REGION Network 62: Falownik P4
   // Sterowaniem pracy z falownika. Sterowanie napędem na pozycji MC
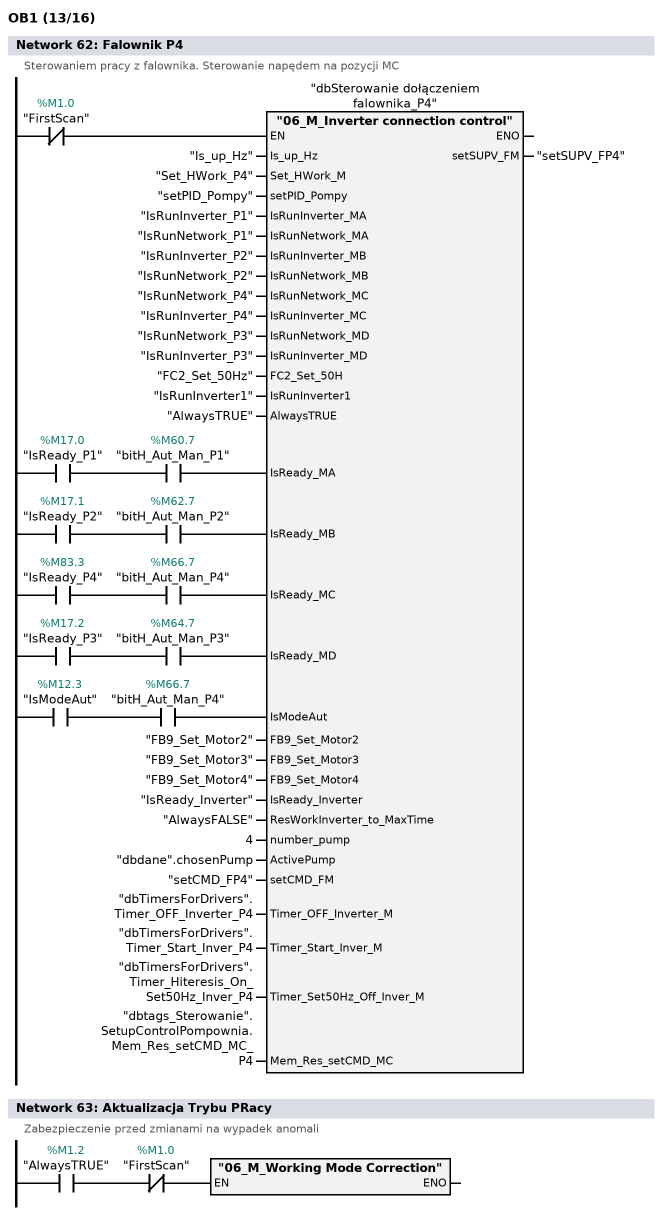
   RUNG wire#powerrail
      I_Contact( "FirstScan" )
      "dbSterowanie dołączeniem falownika_P4"(IsReady_MA := wire#w1, IsReady_MB := wire#w2, IsReady_MC := wire#w3, IsReady_MD := wire#w4, IsModeAut := wire#w5, Is_up_Hz := "Is_up_Hz", Set_HWork_M := "Set_HWork_P4", setPID_Pompy := "setPID_Pompy", IsRunInverter_MA := "IsRunInverter_P1", IsRunNetwork_MA := "IsRunNetwork_P1", IsRunInverter_MB := "IsRunInverter_P2", IsRunNetwork_MB := "IsRunNetwork_P2", IsRunNetwork_MC := "IsRunNetwork_P4", IsRunInverter_MC := "IsRunInverter_P4", IsRunNetwork_MD := "IsRunNetwork_P3", IsRunInverter_MD := "IsRunInverter_P3", FC2_Set_50H := "FC2_Set_50Hz", IsRunInverter1 := "IsRunInverter1", AlwaysTRUE := "AlwaysTRUE", FB9_Set_Motor2 := "FB9_Set_Motor2", FB9_Set_Motor3 := "FB9_Set_Motor3", FB9_Set_Motor4 := "FB9_Set_Motor4", IsReady_Inverter := "IsReady_Inverter", ResWorkInverter_to_MaxTime := "AlwaysFALSE", number_pump := 4, ActivePump := "dbdane".chosenPump, setCMD_FM := "setCMD_FP4", Timer_OFF_Inverter_M := "dbTimersForDrivers".Timer_OFF_Inverter_P4, Timer_Start_Inver_M := "dbTimersForDrivers".Timer_Start_Inver_P4, Timer_Set50Hz_Off_Inver_M := "dbTimersForDrivers".Timer_Hiteresis_On_Set50Hz_Inver_P4, Mem_Res_setCMD_MC := "dbtags_Sterowanie".SetupControlPompownia.Mem_Res_setCMD_MC_P4, setSUPV_FM => "setSUPV_FP4")
   END_RUNG
   RUNG wire#powerrail
      Contact( "IsReady_P1" )
      Contact( "bitH_Aut_Man_P1" )
   END_RUNG wire#w1
   RUNG wire#powerrail
      Contact( "IsReady_P2" )
      Contact( "bitH_Aut_Man_P2" )
   END_RUNG wire#w2
   RUNG wire#powerrail
      Contact( "IsReady_P4" )
      Contact( "bitH_Aut_Man_P4" )
   END_RUNG wire#w3
   RUNG wire#powerrail
      Contact( "IsReady_P3" )
      Contact( "bitH_Aut_Man_P3" )
   END_RUNG wire#w4
   RUNG wire#powerrail
      Contact( "IsModeAut" )
      Contact( "bitH_Aut_Man_P4" )
   END_RUNG wire#w5
   // the same network as SCL:
   IF NOT "FirstScan" THEN
       "dbSterowanie dołączeniem falownika_P4"(Is_up_Hz := "Is_up_Hz",   // "06_M_Inverter connection control"
                               Set_HWork_M := "Set_HWork_P4",
                               setPID_Pompy := "setPID_Pompy",
                               IsRunInverter_MA := "IsRunInverter_P1",
                               IsRunNetwork_MA := "IsRunNetwork_P1",
                               IsRunInverter_MB := "IsRunInverter_P2",
                               IsRunNetwork_MB := "IsRunNetwork_P2",
                               IsRunNetwork_MC := "IsRunNetwork_P4",
                               IsRunInverter_MC := "IsRunInverter_P4",
                               IsRunNetwork_MD := "IsRunNetwork_P3",
                               IsRunInverter_MD := "IsRunInverter_P3",
                               FC2_Set_50H := "FC2_Set_50Hz",
                               IsRunInverter1 := "IsRunInverter1",
                               AlwaysTRUE := "AlwaysTRUE",
                               IsReady_MA := "IsReady_P1" AND "bitH_Aut_Man_P1",
                               IsReady_MB := "IsReady_P2" AND "bitH_Aut_Man_P2",
                               IsReady_MC := "IsReady_P4" AND "bitH_Aut_Man_P4",
                               IsReady_MD := "IsReady_P3" AND "bitH_Aut_Man_P3",
                               IsModeAut := "IsModeAut" AND "bitH_Aut_Man_P4",
                               FB9_Set_Motor2 := "FB9_Set_Motor2",
                               FB9_Set_Motor3 := "FB9_Set_Motor3",
                               FB9_Set_Motor4 := "FB9_Set_Motor4",
                               IsReady_Inverter := "IsReady_Inverter",
                               ResWorkInverter_to_MaxTime := "AlwaysFALSE",
                               number_pump := 4,
                               ActivePump := "dbdane".chosenPump,
                               setCMD_FM := "setCMD_FP4",
                               Timer_OFF_Inverter_M := "dbTimersForDrivers".Timer_OFF_Inverter_P4,
                               Timer_Start_Inver_M := "dbTimersForDrivers".Timer_Start_Inver_P4,
                               Timer_Set50Hz_Off_Inver_M := "dbTimersForDrivers".Timer_Hiteresis_On_Set50Hz_Inver_P4,
                               Mem_Res_setCMD_MC := "dbtags_Sterowanie".SetupControlPompownia.Mem_Res_setCMD_MC_P4,
                               setSUPV_FM => "setSUPV_FP4");
   END_IF;
END_REGION

REGION Network 63: Aktualizacja Trybu PRacy
   // Zabezpieczenie przed zmianami na wypadek anomali
   RUNG wire#powerrail
      Contact( "AlwaysTRUE" )
      I_Contact( "FirstScan" )
      "06_M_Working Mode Correction"()
   END_RUNG
   // the same network as SCL:
   IF "AlwaysTRUE" AND NOT "FirstScan" THEN "06_M_Working Mode Correction"(); END_IF;
END_REGION

REGION Network 64: Sterowanie falownikiem
   // Sterowanie załaczaniem falownika
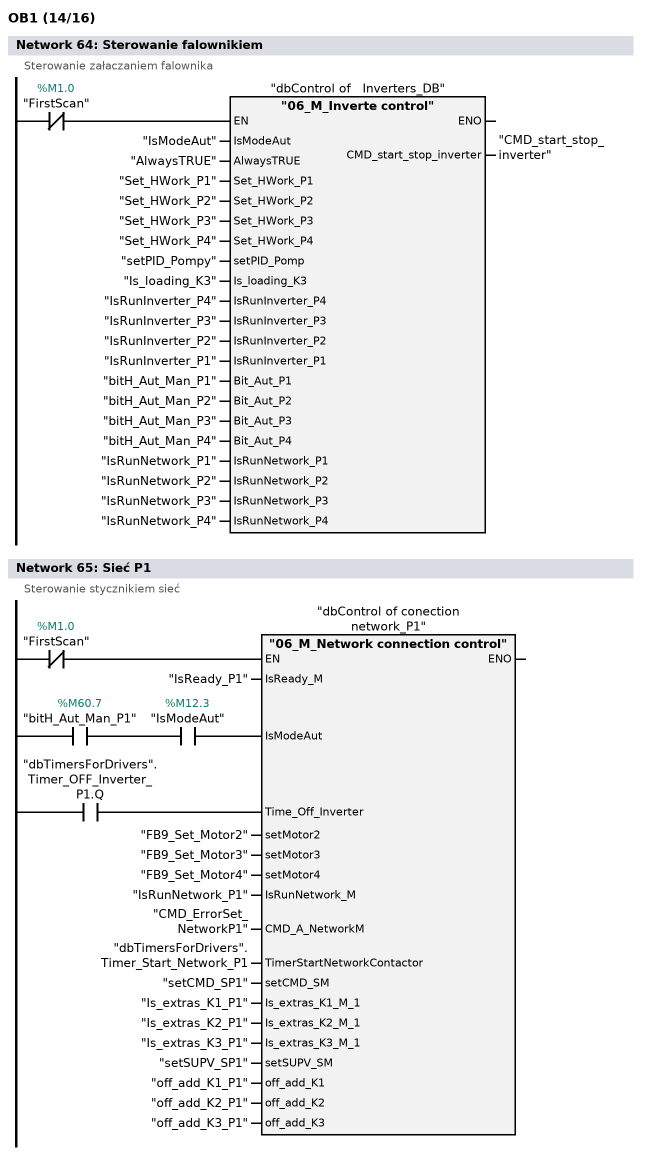
   RUNG wire#powerrail
      I_Contact( "FirstScan" )
      "dbControl of   Inverters_DB"(IsModeAut := "IsModeAut", AlwaysTRUE := "AlwaysTRUE", Set_HWork_P1 := "Set_HWork_P1", Set_HWork_P2 := "Set_HWork_P2", Set_HWork_P3 := "Set_HWork_P3", Set_HWork_P4 := "Set_HWork_P4", setPID_Pomp := "setPID_Pompy", Is_loading_K3 := "Is_loading_K3", IsRunInverter_P4 := "IsRunInverter_P4", IsRunInverter_P3 := "IsRunInverter_P3", IsRunInverter_P2 := "IsRunInverter_P2", IsRunInverter_P1 := "IsRunInverter_P1", Bit_Aut_P1 := "bitH_Aut_Man_P1", Bit_Aut_P2 := "bitH_Aut_Man_P2", Bit_Aut_P3 := "bitH_Aut_Man_P3", Bit_Aut_P4 := "bitH_Aut_Man_P4", IsRunNetwork_P1 := "IsRunNetwork_P1", IsRunNetwork_P2 := "IsRunNetwork_P2", IsRunNetwork_P3 := "IsRunNetwork_P3", IsRunNetwork_P4 := "IsRunNetwork_P4", CMD_start_stop_inverter => "CMD_start_stop_inverter")
   END_RUNG
   // the same network as SCL:
   IF NOT "FirstScan" THEN
       "dbControl of   Inverters_DB"(IsModeAut := "IsModeAut",   // "06_M_Inverte control"
                               AlwaysTRUE := "AlwaysTRUE",
                               Set_HWork_P1 := "Set_HWork_P1",
                               Set_HWork_P2 := "Set_HWork_P2",
                               Set_HWork_P3 := "Set_HWork_P3",
                               Set_HWork_P4 := "Set_HWork_P4",
                               setPID_Pomp := "setPID_Pompy",
                               Is_loading_K3 := "Is_loading_K3",
                               IsRunInverter_P4 := "IsRunInverter_P4",
                               IsRunInverter_P3 := "IsRunInverter_P3",
                               IsRunInverter_P2 := "IsRunInverter_P2",
                               IsRunInverter_P1 := "IsRunInverter_P1",
                               Bit_Aut_P1 := "bitH_Aut_Man_P1",
                               Bit_Aut_P2 := "bitH_Aut_Man_P2",
                               Bit_Aut_P3 := "bitH_Aut_Man_P3",
                               Bit_Aut_P4 := "bitH_Aut_Man_P4",
                               IsRunNetwork_P1 := "IsRunNetwork_P1",
                               IsRunNetwork_P2 := "IsRunNetwork_P2",
                               IsRunNetwork_P3 := "IsRunNetwork_P3",
                               IsRunNetwork_P4 := "IsRunNetwork_P4",
                               CMD_start_stop_inverter => "CMD_start_stop_inverter");
   END_IF;
END_REGION

REGION Network 65: Sieć P1
   // Sterowanie stycznikiem sieć
   RUNG wire#powerrail
      I_Contact( "FirstScan" )
      "dbControl of conection network_P1"(IsModeAut := wire#w1, Time_Off_Inverter := wire#w2, IsReady_M := "IsReady_P1", setMotor2 := "FB9_Set_Motor2", setMotor3 := "FB9_Set_Motor3", setMotor4 := "FB9_Set_Motor4", IsRunNetwork_M := "IsRunNetwork_P1", CMD_A_NetworkM := "CMD_ErrorSet_NetworkP1", TimerStartNetworkContactor := "dbTimersForDrivers".Timer_Start_Network_P1, setCMD_SM := "setCMD_SP1", Is_extras_K1_M_1 := "Is_extras_K1_P1", Is_extras_K2_M_1 := "Is_extras_K2_P1", Is_extras_K3_M_1 := "Is_extras_K3_P1", setSUPV_SM := "setSUPV_SP1", off_add_K1 := "off_add_K1_P1", off_add_K2 := "off_add_K2_P1", off_add_K3 := "off_add_K3_P1")
   END_RUNG
   RUNG wire#powerrail
      Contact( "bitH_Aut_Man_P1" )
      Contact( "IsModeAut" )
   END_RUNG wire#w1
   RUNG wire#powerrail
      Contact( "dbTimersForDrivers".Timer_OFF_Inverter_P1.Q )
   END_RUNG wire#w2
   // the same network as SCL:
   IF NOT "FirstScan" THEN
       "dbControl of conection network_P1"(IsReady_M := "IsReady_P1",   // "06_M_Network connection control"
                               IsModeAut := "bitH_Aut_Man_P1" AND "IsModeAut",
                               Time_Off_Inverter := "dbTimersForDrivers".Timer_OFF_Inverter_P1.Q,
                               setMotor2 := "FB9_Set_Motor2",
                               setMotor3 := "FB9_Set_Motor3",
                               setMotor4 := "FB9_Set_Motor4",
                               IsRunNetwork_M := "IsRunNetwork_P1",
                               CMD_A_NetworkM := "CMD_ErrorSet_NetworkP1",
                               TimerStartNetworkContactor := "dbTimersForDrivers".Timer_Start_Network_P1,
                               setCMD_SM := "setCMD_SP1",
                               Is_extras_K1_M_1 := "Is_extras_K1_P1",
                               Is_extras_K2_M_1 := "Is_extras_K2_P1",
                               Is_extras_K3_M_1 := "Is_extras_K3_P1",
                               setSUPV_SM := "setSUPV_SP1",
                               off_add_K1 := "off_add_K1_P1",
                               off_add_K2 := "off_add_K2_P1",
                               off_add_K3 := "off_add_K3_P1");
   END_IF;
END_REGION

REGION Network 66: Sieć P2
   // Sterowanie stycznikiem sieć
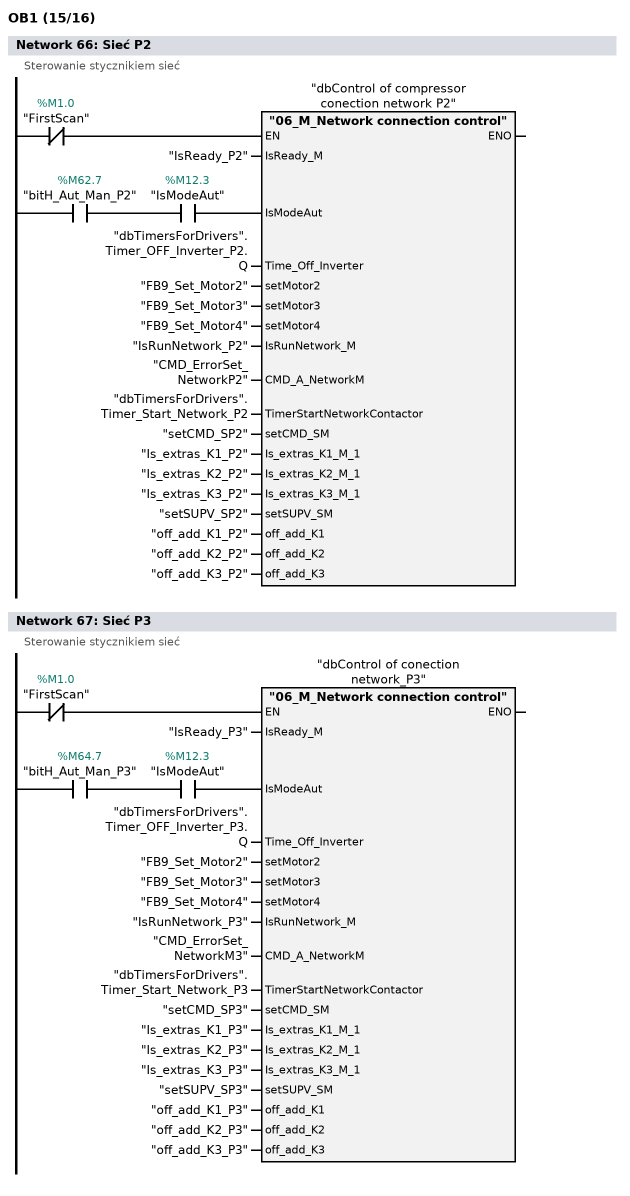
   RUNG wire#powerrail
      I_Contact( "FirstScan" )
      "dbControl of compressor conection network P2"(IsModeAut := wire#w1, IsReady_M := "IsReady_P2", Time_Off_Inverter := "dbTimersForDrivers".Timer_OFF_Inverter_P2.Q, setMotor2 := "FB9_Set_Motor2", setMotor3 := "FB9_Set_Motor3", setMotor4 := "FB9_Set_Motor4", IsRunNetwork_M := "IsRunNetwork_P2", CMD_A_NetworkM := "CMD_ErrorSet_NetworkP2", TimerStartNetworkContactor := "dbTimersForDrivers".Timer_Start_Network_P2, setCMD_SM := "setCMD_SP2", Is_extras_K1_M_1 := "Is_extras_K1_P2", Is_extras_K2_M_1 := "Is_extras_K2_P2", Is_extras_K3_M_1 := "Is_extras_K3_P2", setSUPV_SM := "setSUPV_SP2", off_add_K1 := "off_add_K1_P2", off_add_K2 := "off_add_K2_P2", off_add_K3 := "off_add_K3_P2")
   END_RUNG
   RUNG wire#powerrail
      Contact( "bitH_Aut_Man_P2" )
      Contact( "IsModeAut" )
   END_RUNG wire#w1
   // the same network as SCL:
   IF NOT "FirstScan" THEN
       "dbControl of compressor conection network P2"(IsReady_M := "IsReady_P2",   // "06_M_Network connection control"
                               IsModeAut := "bitH_Aut_Man_P2" AND "IsModeAut",
                               Time_Off_Inverter := "dbTimersForDrivers".Timer_OFF_Inverter_P2.Q,
                               setMotor2 := "FB9_Set_Motor2",
                               setMotor3 := "FB9_Set_Motor3",
                               setMotor4 := "FB9_Set_Motor4",
                               IsRunNetwork_M := "IsRunNetwork_P2",
                               CMD_A_NetworkM := "CMD_ErrorSet_NetworkP2",
                               TimerStartNetworkContactor := "dbTimersForDrivers".Timer_Start_Network_P2,
                               setCMD_SM := "setCMD_SP2",
                               Is_extras_K1_M_1 := "Is_extras_K1_P2",
                               Is_extras_K2_M_1 := "Is_extras_K2_P2",
                               Is_extras_K3_M_1 := "Is_extras_K3_P2",
                               setSUPV_SM := "setSUPV_SP2",
                               off_add_K1 := "off_add_K1_P2",
                               off_add_K2 := "off_add_K2_P2",
                               off_add_K3 := "off_add_K3_P2");
   END_IF;
END_REGION

REGION Network 67: Sieć P3
   // Sterowanie stycznikiem sieć
   RUNG wire#powerrail
      I_Contact( "FirstScan" )
      "dbControl of conection network_P3"(IsModeAut := wire#w1, IsReady_M := "IsReady_P3", Time_Off_Inverter := "dbTimersForDrivers".Timer_OFF_Inverter_P3.Q, setMotor2 := "FB9_Set_Motor2", setMotor3 := "FB9_Set_Motor3", setMotor4 := "FB9_Set_Motor4", IsRunNetwork_M := "IsRunNetwork_P3", CMD_A_NetworkM := "CMD_ErrorSet_NetworkM3", TimerStartNetworkContactor := "dbTimersForDrivers".Timer_Start_Network_P3, setCMD_SM := "setCMD_SP3", Is_extras_K1_M_1 := "Is_extras_K1_P3", Is_extras_K2_M_1 := "Is_extras_K2_P3", Is_extras_K3_M_1 := "Is_extras_K3_P3", setSUPV_SM := "setSUPV_SP3", off_add_K1 := "off_add_K1_P3", off_add_K2 := "off_add_K2_P3", off_add_K3 := "off_add_K3_P3")
   END_RUNG
   RUNG wire#powerrail
      Contact( "bitH_Aut_Man_P3" )
      Contact( "IsModeAut" )
   END_RUNG wire#w1
   // the same network as SCL:
   IF NOT "FirstScan" THEN
       "dbControl of conection network_P3"(IsReady_M := "IsReady_P3",   // "06_M_Network connection control"
                               IsModeAut := "bitH_Aut_Man_P3" AND "IsModeAut",
                               Time_Off_Inverter := "dbTimersForDrivers".Timer_OFF_Inverter_P3.Q,
                               setMotor2 := "FB9_Set_Motor2",
                               setMotor3 := "FB9_Set_Motor3",
                               setMotor4 := "FB9_Set_Motor4",
                               IsRunNetwork_M := "IsRunNetwork_P3",
                               CMD_A_NetworkM := "CMD_ErrorSet_NetworkM3",
                               TimerStartNetworkContactor := "dbTimersForDrivers".Timer_Start_Network_P3,
                               setCMD_SM := "setCMD_SP3",
                               Is_extras_K1_M_1 := "Is_extras_K1_P3",
                               Is_extras_K2_M_1 := "Is_extras_K2_P3",
                               Is_extras_K3_M_1 := "Is_extras_K3_P3",
                               setSUPV_SM := "setSUPV_SP3",
                               off_add_K1 := "off_add_K1_P3",
                               off_add_K2 := "off_add_K2_P3",
                               off_add_K3 := "off_add_K3_P3");
   END_IF;
END_REGION

REGION Network 68: Sieć P4
   // !!!!!!!!!!!!!!!!!!!!! ------------------ Brak pompy --------------------------!!!!!!!!!!!!!!!!!!!!!!!!!!!!!!!
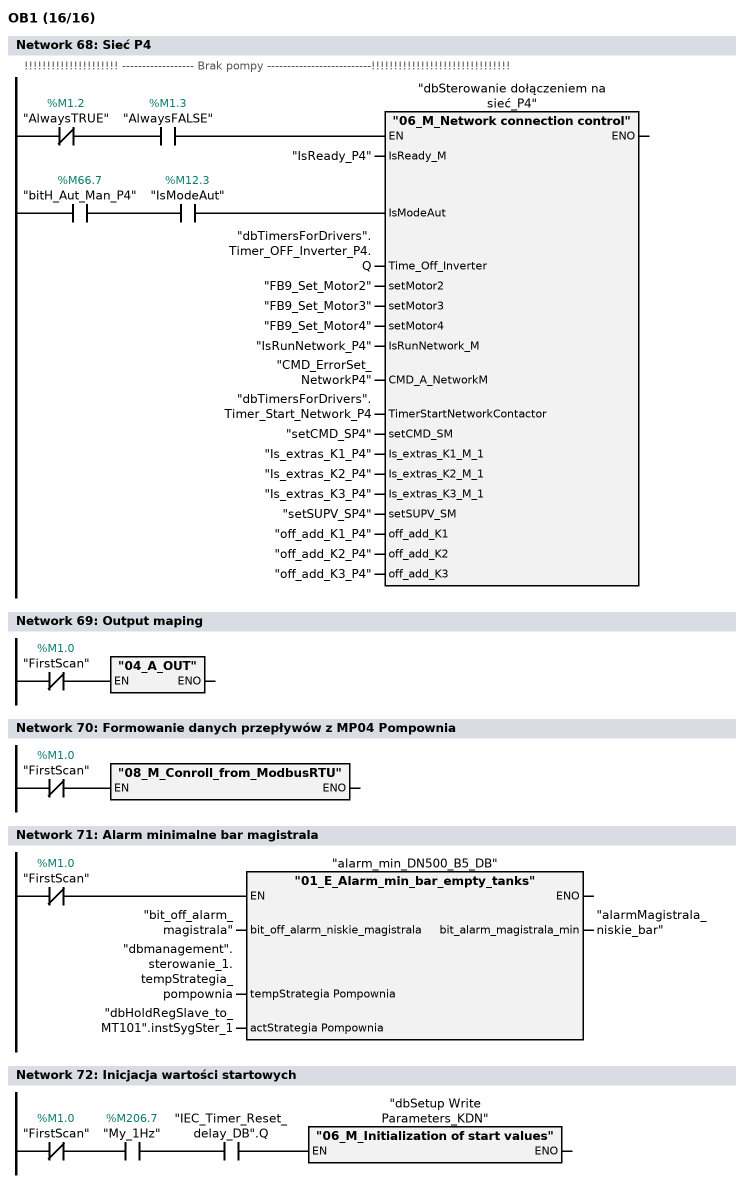
   RUNG wire#powerrail
      I_Contact( "AlwaysTRUE" )
      Contact( "AlwaysFALSE" )
      "dbSterowanie dołączeniem na sieć_P4"(IsModeAut := wire#w1, IsReady_M := "IsReady_P4", Time_Off_Inverter := "dbTimersForDrivers".Timer_OFF_Inverter_P4.Q, setMotor2 := "FB9_Set_Motor2", setMotor3 := "FB9_Set_Motor3", setMotor4 := "FB9_Set_Motor4", IsRunNetwork_M := "IsRunNetwork_P4", CMD_A_NetworkM := "CMD_ErrorSet_NetworkP4", TimerStartNetworkContactor := "dbTimersForDrivers".Timer_Start_Network_P4, setCMD_SM := "setCMD_SP4", Is_extras_K1_M_1 := "Is_extras_K1_P4", Is_extras_K2_M_1 := "Is_extras_K2_P4", Is_extras_K3_M_1 := "Is_extras_K3_P4", setSUPV_SM := "setSUPV_SP4", off_add_K1 := "off_add_K1_P4", off_add_K2 := "off_add_K2_P4", off_add_K3 := "off_add_K3_P4")
   END_RUNG
   RUNG wire#powerrail
      Contact( "bitH_Aut_Man_P4" )
      Contact( "IsModeAut" )
   END_RUNG wire#w1
   // the same network as SCL:
   IF NOT "AlwaysTRUE" AND "AlwaysFALSE" THEN
       "dbSterowanie dołączeniem na sieć_P4"(IsReady_M := "IsReady_P4",   // "06_M_Network connection control"
                               IsModeAut := "bitH_Aut_Man_P4" AND "IsModeAut",
                               Time_Off_Inverter := "dbTimersForDrivers".Timer_OFF_Inverter_P4.Q,
                               setMotor2 := "FB9_Set_Motor2",
                               setMotor3 := "FB9_Set_Motor3",
                               setMotor4 := "FB9_Set_Motor4",
                               IsRunNetwork_M := "IsRunNetwork_P4",
                               CMD_A_NetworkM := "CMD_ErrorSet_NetworkP4",
                               TimerStartNetworkContactor := "dbTimersForDrivers".Timer_Start_Network_P4,
                               setCMD_SM := "setCMD_SP4",
                               Is_extras_K1_M_1 := "Is_extras_K1_P4",
                               Is_extras_K2_M_1 := "Is_extras_K2_P4",
                               Is_extras_K3_M_1 := "Is_extras_K3_P4",
                               setSUPV_SM := "setSUPV_SP4",
                               off_add_K1 := "off_add_K1_P4",
                               off_add_K2 := "off_add_K2_P4",
                               off_add_K3 := "off_add_K3_P4");
   END_IF;
END_REGION

REGION Network 69: Output maping
   RUNG wire#powerrail
      I_Contact( "FirstScan" )
      "04_A_OUT"()
   END_RUNG
   // the same network as SCL:
   IF NOT "FirstScan" THEN "04_A_OUT"(); END_IF;
END_REGION

REGION Network 70: Formowanie danych przepływów z MP04 Pompownia
   RUNG wire#powerrail
      I_Contact( "FirstScan" )
      "08_M_Conroll_from_ModbusRTU"()
   END_RUNG
   // the same network as SCL:
   IF NOT "FirstScan" THEN "08_M_Conroll_from_ModbusRTU"(); END_IF;
END_REGION

REGION Network 71: Alarm minimalne bar magistrala
   RUNG wire#powerrail
      I_Contact( "FirstScan" )
      "alarm_min_DN500_B5_DB"(bit_off_alarm_niskie_magistrala := "bit_off_alarm_magistrala", "tempStrategia Pompownia" := "dbmanagement".sterowanie_1.tempStrategia_pompownia, "actStrategia Pompownia" := "dbHoldRegSlave_to_MT101".instSygSter_1, bit_alarm_magistrala_min => "alarmMagistrala_niskie_bar")
   END_RUNG
   // the same network as SCL:
   IF NOT "FirstScan" THEN
       "alarm_min_DN500_B5_DB"(bit_off_alarm_niskie_magistrala := "bit_off_alarm_magistrala",   // "01_E_Alarm_min_bar_empty_tanks"
                               "tempStrategia Pompownia" := "dbmanagement".sterowanie_1.tempStrategia_pompownia,
                               "actStrategia Pompownia" := "dbHoldRegSlave_to_MT101".instSygSter_1,
                               bit_alarm_magistrala_min => "alarmMagistrala_niskie_bar");
   END_IF;
END_REGION

REGION Network 72: Inicjacja wartości startowych
   RUNG wire#powerrail
      I_Contact( "FirstScan" )
      Contact( "My_1Hz" )
      Contact( "IEC_Timer_Reset_delay_DB".Q )
      "dbSetup Write Parameters_KDN"()
   END_RUNG
   // the same network as SCL:
   IF NOT "FirstScan" AND "My_1Hz" AND "IEC_Timer_Reset_delay_DB".Q THEN
       "dbSetup Write Parameters_KDN"();   // "06_M_Initialization of start values"
   END_IF;
END_REGION
END_ORGANIZATION_BLOCK

FUNCTION "02_R_RTC" : Void   // FC44, LAD
{ S7_Optimized_Access := 'TRUE' }
VERSION : 0.1
// stored: AutoNumber true, IsIECCheckEnabled false, SetENOAutomatically false, UDAEnableTagReadback false
   VAR_TEMP   // added for the SCL form of the ladder/FBD networks
      _w1 : Bool;
      _w2 : Bool;
   END_VAR
BEGIN

REGION Network 1
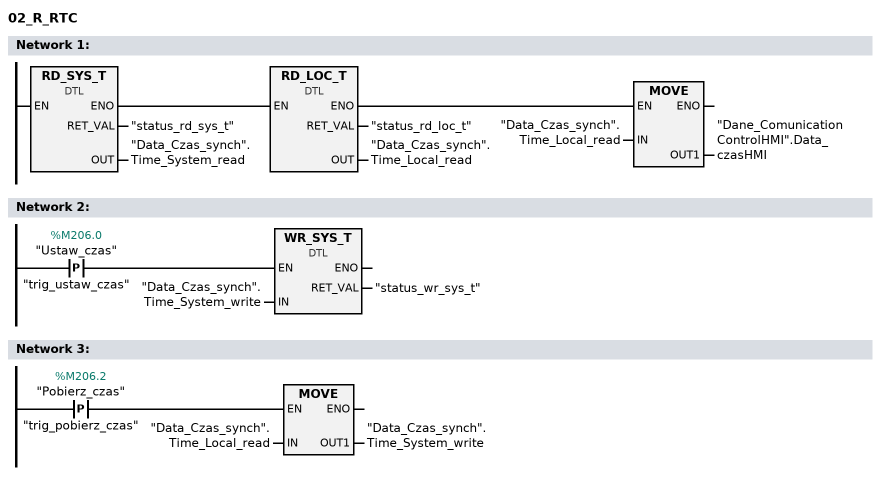
   RUNG wire#powerrail
      { S7_Templates := "date_type := DTL" } RD_SYS_T(RET_VAL => "status_rd_sys_t", OUT => "Data_Czas_synch".Time_System_read)
      { S7_Templates := "date_type := DTL" } RD_LOC_T(RET_VAL => "status_rd_loc_t", OUT => "Data_Czas_synch".Time_Local_read)
      { S7_GenerateENO := "TRUE" } Move(in := "Data_Czas_synch".Time_Local_read, out1 => "Dane_ComunicationControlHMI".Data_czasHMI)
   END_RUNG
   // the same network as SCL:
   "status_rd_sys_t" := RD_SYS_T(OUT => "Data_Czas_synch".Time_System_read, ENO => #_w1);
   "status_rd_loc_t" := RD_LOC_T(EN := #_w1, OUT => "Data_Czas_synch".Time_Local_read, ENO => #_w2);
   IF #_w2 THEN "Dane_ComunicationControlHMI".Data_czasHMI := "Data_Czas_synch".Time_Local_read; END_IF;
END_REGION

REGION Network 2
   RUNG wire#powerrail
      P_Contact(operand := "Ustaw_czas", bit := "trig_ustaw_czas")
      { S7_Templates := "date_type := DTL" } WR_SYS_T(IN := "Data_Czas_synch".Time_System_write, RET_VAL => "status_wr_sys_t")
   END_RUNG
   // the same network as SCL:
   #_w1 := "Ustaw_czas" AND NOT "trig_ustaw_czas";   // rising edge of "Ustaw_czas"
   "trig_ustaw_czas" := "Ustaw_czas";
   IF #_w1 THEN "status_wr_sys_t" := WR_SYS_T(IN := "Data_Czas_synch".Time_System_write); END_IF;
END_REGION

REGION Network 3
   RUNG wire#powerrail
      P_Contact(operand := "Pobierz_czas", bit := "trig_pobierz_czas")
      { S7_GenerateENO := "TRUE" } Move(in := "Data_Czas_synch".Time_Local_read, out1 => "Data_Czas_synch".Time_System_write)
   END_RUNG
   // the same network as SCL:
   #_w1 := "Pobierz_czas" AND NOT "trig_pobierz_czas";   // rising edge of "Pobierz_czas"
   "trig_pobierz_czas" := "Pobierz_czas";
   IF #_w1 THEN "Data_Czas_synch".Time_System_write := "Data_Czas_synch".Time_Local_read; END_IF;
END_REGION
END_FUNCTION

FUNCTION "08_C_clear_drive_error" : Void
TITLE = Modbus RTU Master do Slave przetwarzanie 
{ S7_Optimized_Access := 'TRUE' }
AUTHOR : rtecmer
VERSION : 0.1
//Funkcja przetwarz przekazane sygnały kasowania alarmów z mastera Modbus RTU (MT101) i wykonuje operację

BEGIN
	(*
	//=============================================================================
	//(JZWiK S.A Radosław Tecmer)
	//(c)Copyright (2021) All Rights Reserved
	//-----------------------------------------------------------------------------
	//Testowane z:   (system docelowy z  FW 4.2)
	//Pakiet inżynierski:   TIA Portal (V14 Sp1 Update 9)
	//Ograniczenia:  ( - )
	//Wymagania:  (minimalne S7-1200 CPU 1214 FW 3.2 .)
	//Funkcjonalnośc: (Pzetwarzanie sygnałów z MT101 protokołem Modbus RTU. 
	                    Kasowanie alarów)
	//-----------------------------------------------------------------------------
	//Zmainy wprowadzone:
	//Wersja  Data       Osoba wprowadzająca zmiany - ekspert
	//01.00.00 17.11.2021 (Tecmer Radosław - twórca) Pieresza wersja 01.00.00
	//=============================================================================
	*)
	
	//--- Kasowanie Alarmu Napędów
	
	//Ustawienie bitu Reset dla Drive Motor 1
	%DB100.DBX0.6 := %DB100.DBX51.0;
	IF %DB100.DBX1.0 = FALSE AND %DB100.DBX51.0 = TRUE  THEN
	  // ustaw automat
	  %DB100.DBX0.7 := TRUE;
	  // Kasowanie bitu RESET Driver i Modbus bit Reset
	  %DB100.DBX0.0 := FALSE;
	  %DB100.DBX51.0 := False;
	  ;
	END_IF;
	
	//Ustawienie bitu Reset dla Drive Motor 2
	%DB100.DBX2.6 := %DB100.DBX51.1;
	IF %DB100.DBX1.0 = FALSE AND %DB100.DBX51.1 =TRUE  THEN
	  // ustaw automat
	  %DB100.DBX2.7 := TRUE;
	  // Kasowanie bitu RESET Driver i Modbus bit Reset
	  %DB100.DBX2.0 := FALSE;
	  %DB100.DBX51.1 := False;
	  ;
	END_IF;
	
	//Ustawienie bitu Reset dla Drive Motor 3
	%DB100.DBX4.6 := %DB100.DBX51.2;
	IF %DB100.DBX4.0 = FALSE AND  %DB100.DBX51.2 = TRUE THEN
	  // ustaw automat
	  %DB100.DBX4.7 := TRUE;
	  // Kasowanie bitu RESET Driver i Modbus bit Reset
	  %DB100.DBX4.0 := FALSE;
	  %DB100.DBX51.2 := False;
	  ;
	END_IF;
	
	//Ustawienie bitu Reset dla Drive Motor 4
	%DB100.DBX6.6 := %DB100.DBX51.3;
	IF %DB100.DBX6.0 = FALSE AND %DB100.DBX51.3 = TRUE THEN
	  // ustaw automat
	  %DB100.DBX6.7 := TRUE;
	  // Kasowanie bitu RESET Driver i Modbus bit Reset
	  %DB100.DBX6.0 := FALSE;
	  %DB100.DBX51.3 := False;
	  ;
	END_IF;
	
	
	//Ustawienie bitu Reset dla Drive Z11
	%DB100.DBX28.6 := %DB100.DBX50.6;
	IF %DB100.DBX28.0 = FALSE AND %DB100.DBX50.6 = TRUE THEN
	  // ustaw automat
	  %DB100.DBX28.7 := TRUE;
	  // Kasowanie bitu RESET Driver i Modbus bit Reset
	  %DB100.DBX28.0 := FALSE;
	  %DB100.DBX50.6 := False;
	  ;
	END_IF;
	
	
	
	
	
	
	
	
	
	
	
	
	
	
	
	
	
END_FUNCTION

FUNCTION "08_C_Synchroniczna_wymiana_danych_PLC1-PLC2" : Void   // FC61, LAD
TITLE = Wymiana danych
{ S7_Optimized_Access := 'TRUE' }
AUTHOR : rtecmer
VERSION : 0.1
// Funkcja grupuje bloki funkcji służąc wymianie danych HMI - PLC1, HMI-PLC2 i SCADA. Wprowadzanie wartości z poziomu HMI Zbiorniki lub HMI Pompownia czy SCADA jest nadpisywane w docelowym sterowniku. Zmian włónych parametrów układu sterowania pompownią, zbiornikami można dokonywać w dowolnego miejsca.
// stored: AutoNumber true, IsIECCheckEnabled false, SetENOAutomatically false, UDAEnableTagReadback false
   VAR_TEMP   // added for the SCL form of the ladder/FBD networks
      _w1 : Bool;
   END_VAR
BEGIN

REGION Network 2: Detekcja zmiany danych - Poziom napełnienia
   // Wymiana danych między PLC 1, PLC 2, SCADA
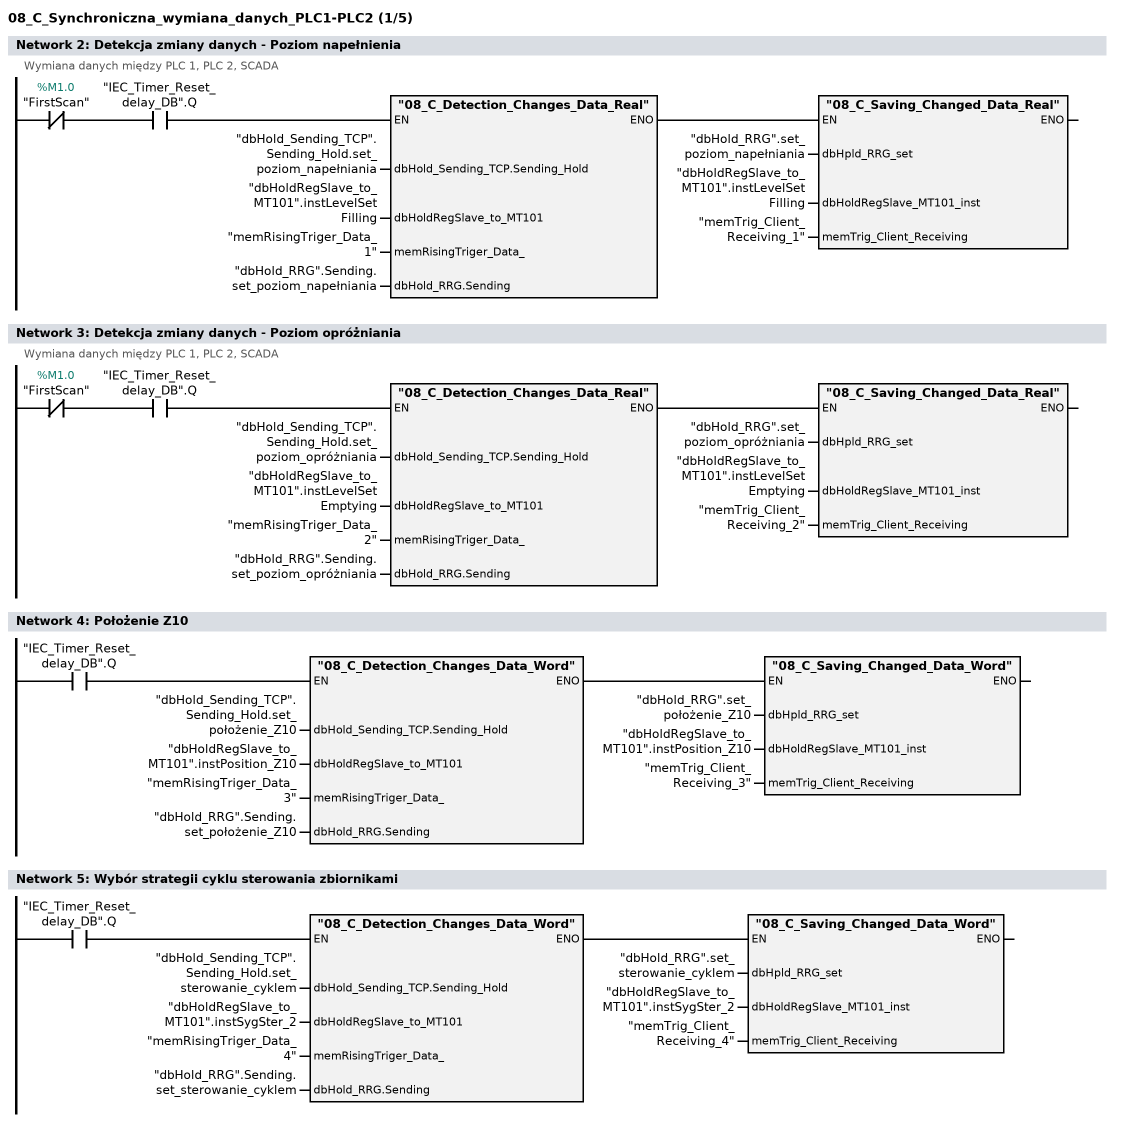
   RUNG wire#powerrail
      I_Contact( "FirstScan" )
      Contact( "IEC_Timer_Reset_delay_DB".Q )
      "08_C_Detection_Changes_Data_Real"("dbHold_Sending_TCP.Sending_Hold" := "dbHold_Sending_TCP".Sending_Hold.set_poziom_napełniania, dbHoldRegSlave_to_MT101 := "dbHoldRegSlave_to_MT101".instLevelSetFilling, memRisingTriger_Data_ := "memRisingTriger_Data_1", "dbHold_RRG.Sending" := "dbHold_RRG".Sending.set_poziom_napełniania)
      "08_C_Saving_Changed_Data_Real"(dbHpld_RRG_set := "dbHold_RRG".set_poziom_napełniania, dbHoldRegSlave_MT101_inst := "dbHoldRegSlave_to_MT101".instLevelSetFilling, memTrig_Client_Receiving := "memTrig_Client_Receiving_1")
   END_RUNG
   // the same network as SCL:
   "08_C_Detection_Changes_Data_Real"(EN := NOT "FirstScan" AND "IEC_Timer_Reset_delay_DB".Q,
                           "dbHold_Sending_TCP.Sending_Hold" := "dbHold_Sending_TCP".Sending_Hold.set_poziom_napełniania,
                           dbHoldRegSlave_to_MT101 := "dbHoldRegSlave_to_MT101".instLevelSetFilling,
                           memRisingTriger_Data_ := "memRisingTriger_Data_1",
                           "dbHold_RRG.Sending" := "dbHold_RRG".Sending.set_poziom_napełniania,
                           ENO => #_w1);
   IF #_w1 THEN
       "08_C_Saving_Changed_Data_Real"(dbHpld_RRG_set := "dbHold_RRG".set_poziom_napełniania,
                               dbHoldRegSlave_MT101_inst := "dbHoldRegSlave_to_MT101".instLevelSetFilling,
                               memTrig_Client_Receiving := "memTrig_Client_Receiving_1");
   END_IF;
END_REGION

REGION Network 3: Detekcja zmiany danych - Poziom opróżniania
   // Wymiana danych między PLC 1, PLC 2, SCADA
   RUNG wire#powerrail
      I_Contact( "FirstScan" )
      Contact( "IEC_Timer_Reset_delay_DB".Q )
      "08_C_Detection_Changes_Data_Real"("dbHold_Sending_TCP.Sending_Hold" := "dbHold_Sending_TCP".Sending_Hold.set_poziom_opróżniania, dbHoldRegSlave_to_MT101 := "dbHoldRegSlave_to_MT101".instLevelSetEmptying, memRisingTriger_Data_ := "memRisingTriger_Data_2", "dbHold_RRG.Sending" := "dbHold_RRG".Sending.set_poziom_opróżniania)
      "08_C_Saving_Changed_Data_Real"(dbHpld_RRG_set := "dbHold_RRG".set_poziom_opróżniania, dbHoldRegSlave_MT101_inst := "dbHoldRegSlave_to_MT101".instLevelSetEmptying, memTrig_Client_Receiving := "memTrig_Client_Receiving_2")
   END_RUNG
   // the same network as SCL:
   "08_C_Detection_Changes_Data_Real"(EN := NOT "FirstScan" AND "IEC_Timer_Reset_delay_DB".Q,
                           "dbHold_Sending_TCP.Sending_Hold" := "dbHold_Sending_TCP".Sending_Hold.set_poziom_opróżniania,
                           dbHoldRegSlave_to_MT101 := "dbHoldRegSlave_to_MT101".instLevelSetEmptying,
                           memRisingTriger_Data_ := "memRisingTriger_Data_2",
                           "dbHold_RRG.Sending" := "dbHold_RRG".Sending.set_poziom_opróżniania,
                           ENO => #_w1);
   IF #_w1 THEN
       "08_C_Saving_Changed_Data_Real"(dbHpld_RRG_set := "dbHold_RRG".set_poziom_opróżniania,
                               dbHoldRegSlave_MT101_inst := "dbHoldRegSlave_to_MT101".instLevelSetEmptying,
                               memTrig_Client_Receiving := "memTrig_Client_Receiving_2");
   END_IF;
END_REGION

REGION Network 4: Położenie Z10
   RUNG wire#powerrail
      Contact( "IEC_Timer_Reset_delay_DB".Q )
      "08_C_Detection_Changes_Data_Word"("dbHold_Sending_TCP.Sending_Hold" := "dbHold_Sending_TCP".Sending_Hold.set_położenie_Z10, dbHoldRegSlave_to_MT101 := "dbHoldRegSlave_to_MT101".instPosition_Z10, memRisingTriger_Data_ := "memRisingTriger_Data_3", "dbHold_RRG.Sending" := "dbHold_RRG".Sending.set_położenie_Z10)
      "08_C_Saving_Changed_Data_Word"(dbHpld_RRG_set := "dbHold_RRG".set_położenie_Z10, dbHoldRegSlave_MT101_inst := "dbHoldRegSlave_to_MT101".instPosition_Z10, memTrig_Client_Receiving := "memTrig_Client_Receiving_3")
   END_RUNG
   // the same network as SCL:
   "08_C_Detection_Changes_Data_Word"(EN := "IEC_Timer_Reset_delay_DB".Q,
                           "dbHold_Sending_TCP.Sending_Hold" := "dbHold_Sending_TCP".Sending_Hold.set_położenie_Z10,
                           dbHoldRegSlave_to_MT101 := "dbHoldRegSlave_to_MT101".instPosition_Z10,
                           memRisingTriger_Data_ := "memRisingTriger_Data_3",
                           "dbHold_RRG.Sending" := "dbHold_RRG".Sending.set_położenie_Z10,
                           ENO => #_w1);
   IF #_w1 THEN
       "08_C_Saving_Changed_Data_Word"(dbHpld_RRG_set := "dbHold_RRG".set_położenie_Z10,
                               dbHoldRegSlave_MT101_inst := "dbHoldRegSlave_to_MT101".instPosition_Z10,
                               memTrig_Client_Receiving := "memTrig_Client_Receiving_3");
   END_IF;
END_REGION

REGION Network 5: Wybór strategii cyklu sterowania zbiornikami
   RUNG wire#powerrail
      Contact( "IEC_Timer_Reset_delay_DB".Q )
      "08_C_Detection_Changes_Data_Word"("dbHold_Sending_TCP.Sending_Hold" := "dbHold_Sending_TCP".Sending_Hold.set_sterowanie_cyklem, dbHoldRegSlave_to_MT101 := "dbHoldRegSlave_to_MT101".instSygSter_2, memRisingTriger_Data_ := "memRisingTriger_Data_4", "dbHold_RRG.Sending" := "dbHold_RRG".Sending.set_sterowanie_cyklem)
      "08_C_Saving_Changed_Data_Word"(dbHpld_RRG_set := "dbHold_RRG".set_sterowanie_cyklem, dbHoldRegSlave_MT101_inst := "dbHoldRegSlave_to_MT101".instSygSter_2, memTrig_Client_Receiving := "memTrig_Client_Receiving_4")
   END_RUNG
   // the same network as SCL:
   "08_C_Detection_Changes_Data_Word"(EN := "IEC_Timer_Reset_delay_DB".Q,
                           "dbHold_Sending_TCP.Sending_Hold" := "dbHold_Sending_TCP".Sending_Hold.set_sterowanie_cyklem,
                           dbHoldRegSlave_to_MT101 := "dbHoldRegSlave_to_MT101".instSygSter_2,
                           memRisingTriger_Data_ := "memRisingTriger_Data_4",
                           "dbHold_RRG.Sending" := "dbHold_RRG".Sending.set_sterowanie_cyklem,
                           ENO => #_w1);
   IF #_w1 THEN
       "08_C_Saving_Changed_Data_Word"(dbHpld_RRG_set := "dbHold_RRG".set_sterowanie_cyklem,
                               dbHoldRegSlave_MT101_inst := "dbHoldRegSlave_to_MT101".instSygSter_2,
                               memTrig_Client_Receiving := "memTrig_Client_Receiving_4");
   END_IF;
END_REGION

REGION Network 6: Godzina napełniania start
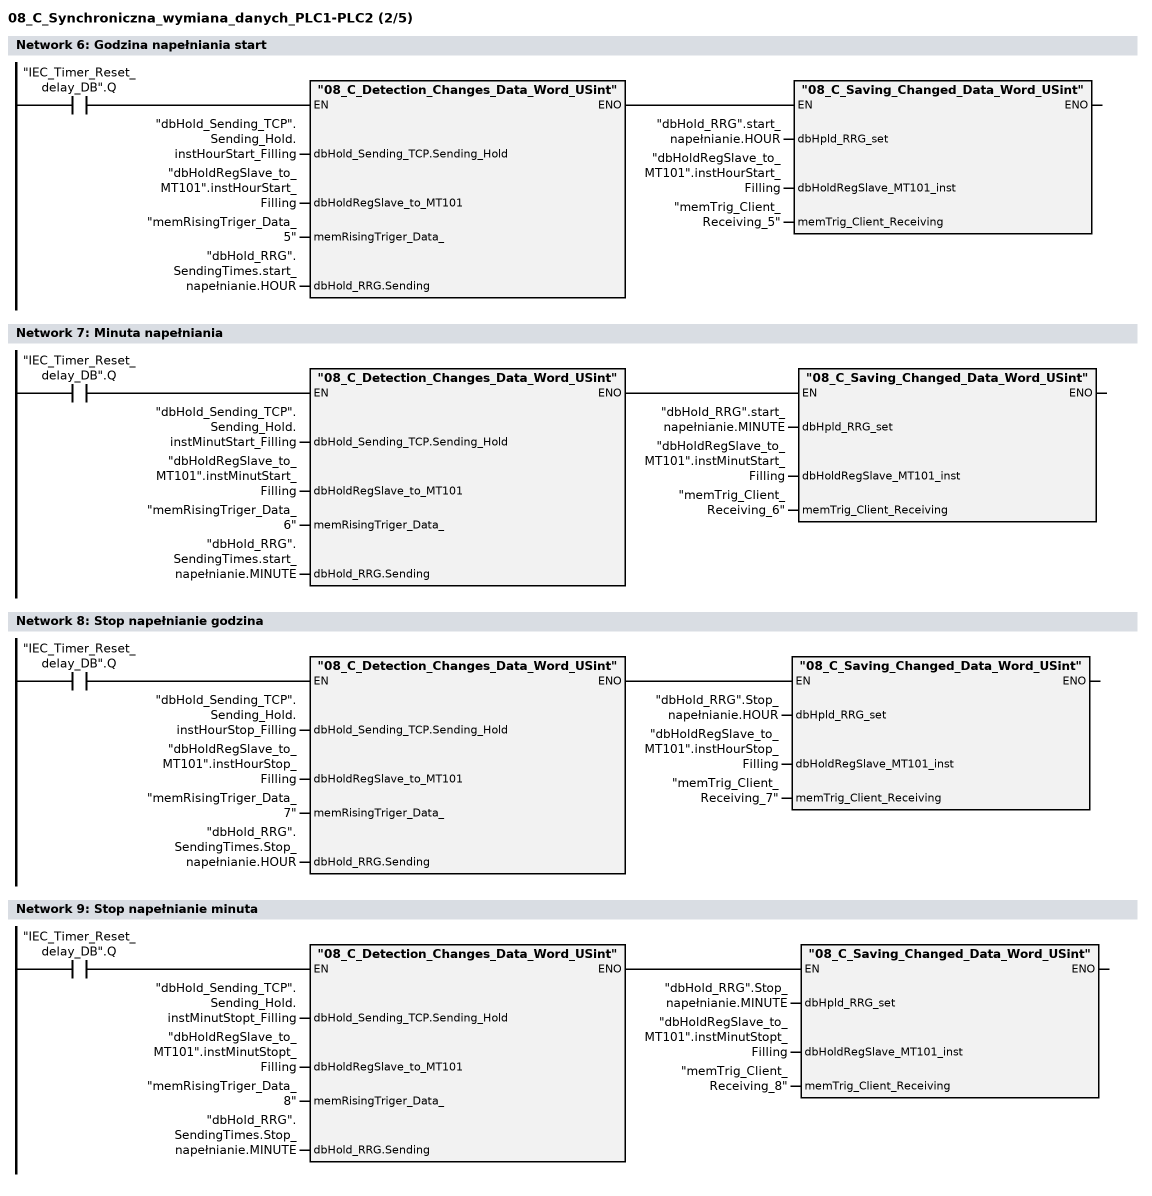
   RUNG wire#powerrail
      Contact( "IEC_Timer_Reset_delay_DB".Q )
      "08_C_Detection_Changes_Data_Word_USint"("dbHold_Sending_TCP.Sending_Hold" := "dbHold_Sending_TCP".Sending_Hold.instHourStart_Filling, dbHoldRegSlave_to_MT101 := "dbHoldRegSlave_to_MT101".instHourStart_Filling, memRisingTriger_Data_ := "memRisingTriger_Data_5", "dbHold_RRG.Sending" := "dbHold_RRG".SendingTimes.start_napełnianie.HOUR)
      "08_C_Saving_Changed_Data_Word_USint"(dbHpld_RRG_set := "dbHold_RRG".start_napełnianie.HOUR, dbHoldRegSlave_MT101_inst := "dbHoldRegSlave_to_MT101".instHourStart_Filling, memTrig_Client_Receiving := "memTrig_Client_Receiving_5")
   END_RUNG
   // the same network as SCL:
   "08_C_Detection_Changes_Data_Word_USint"(EN := "IEC_Timer_Reset_delay_DB".Q,
                           "dbHold_Sending_TCP.Sending_Hold" := "dbHold_Sending_TCP".Sending_Hold.instHourStart_Filling,
                           dbHoldRegSlave_to_MT101 := "dbHoldRegSlave_to_MT101".instHourStart_Filling,
                           memRisingTriger_Data_ := "memRisingTriger_Data_5",
                           "dbHold_RRG.Sending" := "dbHold_RRG".SendingTimes.start_napełnianie.HOUR,
                           ENO => #_w1);
   IF #_w1 THEN
       "08_C_Saving_Changed_Data_Word_USint"(dbHpld_RRG_set := "dbHold_RRG".start_napełnianie.HOUR,
                               dbHoldRegSlave_MT101_inst := "dbHoldRegSlave_to_MT101".instHourStart_Filling,
                               memTrig_Client_Receiving := "memTrig_Client_Receiving_5");
   END_IF;
END_REGION

REGION Network 7: Minuta napełniania
   RUNG wire#powerrail
      Contact( "IEC_Timer_Reset_delay_DB".Q )
      "08_C_Detection_Changes_Data_Word_USint"("dbHold_Sending_TCP.Sending_Hold" := "dbHold_Sending_TCP".Sending_Hold.instMinutStart_Filling, dbHoldRegSlave_to_MT101 := "dbHoldRegSlave_to_MT101".instMinutStart_Filling, memRisingTriger_Data_ := "memRisingTriger_Data_6", "dbHold_RRG.Sending" := "dbHold_RRG".SendingTimes.start_napełnianie.MINUTE)
      "08_C_Saving_Changed_Data_Word_USint"(dbHpld_RRG_set := "dbHold_RRG".start_napełnianie.MINUTE, dbHoldRegSlave_MT101_inst := "dbHoldRegSlave_to_MT101".instMinutStart_Filling, memTrig_Client_Receiving := "memTrig_Client_Receiving_6")
   END_RUNG
   // the same network as SCL:
   "08_C_Detection_Changes_Data_Word_USint"(EN := "IEC_Timer_Reset_delay_DB".Q,
                           "dbHold_Sending_TCP.Sending_Hold" := "dbHold_Sending_TCP".Sending_Hold.instMinutStart_Filling,
                           dbHoldRegSlave_to_MT101 := "dbHoldRegSlave_to_MT101".instMinutStart_Filling,
                           memRisingTriger_Data_ := "memRisingTriger_Data_6",
                           "dbHold_RRG.Sending" := "dbHold_RRG".SendingTimes.start_napełnianie.MINUTE,
                           ENO => #_w1);
   IF #_w1 THEN
       "08_C_Saving_Changed_Data_Word_USint"(dbHpld_RRG_set := "dbHold_RRG".start_napełnianie.MINUTE,
                               dbHoldRegSlave_MT101_inst := "dbHoldRegSlave_to_MT101".instMinutStart_Filling,
                               memTrig_Client_Receiving := "memTrig_Client_Receiving_6");
   END_IF;
END_REGION

REGION Network 8: Stop napełnianie godzina
   RUNG wire#powerrail
      Contact( "IEC_Timer_Reset_delay_DB".Q )
      "08_C_Detection_Changes_Data_Word_USint"("dbHold_Sending_TCP.Sending_Hold" := "dbHold_Sending_TCP".Sending_Hold.instHourStop_Filling, dbHoldRegSlave_to_MT101 := "dbHoldRegSlave_to_MT101".instHourStop_Filling, memRisingTriger_Data_ := "memRisingTriger_Data_7", "dbHold_RRG.Sending" := "dbHold_RRG".SendingTimes.Stop_napełnianie.HOUR)
      "08_C_Saving_Changed_Data_Word_USint"(dbHpld_RRG_set := "dbHold_RRG".Stop_napełnianie.HOUR, dbHoldRegSlave_MT101_inst := "dbHoldRegSlave_to_MT101".instHourStop_Filling, memTrig_Client_Receiving := "memTrig_Client_Receiving_7")
   END_RUNG
   // the same network as SCL:
   "08_C_Detection_Changes_Data_Word_USint"(EN := "IEC_Timer_Reset_delay_DB".Q,
                           "dbHold_Sending_TCP.Sending_Hold" := "dbHold_Sending_TCP".Sending_Hold.instHourStop_Filling,
                           dbHoldRegSlave_to_MT101 := "dbHoldRegSlave_to_MT101".instHourStop_Filling,
                           memRisingTriger_Data_ := "memRisingTriger_Data_7",
                           "dbHold_RRG.Sending" := "dbHold_RRG".SendingTimes.Stop_napełnianie.HOUR,
                           ENO => #_w1);
   IF #_w1 THEN
       "08_C_Saving_Changed_Data_Word_USint"(dbHpld_RRG_set := "dbHold_RRG".Stop_napełnianie.HOUR,
                               dbHoldRegSlave_MT101_inst := "dbHoldRegSlave_to_MT101".instHourStop_Filling,
                               memTrig_Client_Receiving := "memTrig_Client_Receiving_7");
   END_IF;
END_REGION

REGION Network 9: Stop napełnianie minuta
   RUNG wire#powerrail
      Contact( "IEC_Timer_Reset_delay_DB".Q )
      "08_C_Detection_Changes_Data_Word_USint"("dbHold_Sending_TCP.Sending_Hold" := "dbHold_Sending_TCP".Sending_Hold.instMinutStopt_Filling, dbHoldRegSlave_to_MT101 := "dbHoldRegSlave_to_MT101".instMinutStopt_Filling, memRisingTriger_Data_ := "memRisingTriger_Data_8", "dbHold_RRG.Sending" := "dbHold_RRG".SendingTimes.Stop_napełnianie.MINUTE)
      "08_C_Saving_Changed_Data_Word_USint"(dbHpld_RRG_set := "dbHold_RRG".Stop_napełnianie.MINUTE, dbHoldRegSlave_MT101_inst := "dbHoldRegSlave_to_MT101".instMinutStopt_Filling, memTrig_Client_Receiving := "memTrig_Client_Receiving_8")
   END_RUNG
   // the same network as SCL:
   "08_C_Detection_Changes_Data_Word_USint"(EN := "IEC_Timer_Reset_delay_DB".Q,
                           "dbHold_Sending_TCP.Sending_Hold" := "dbHold_Sending_TCP".Sending_Hold.instMinutStopt_Filling,
                           dbHoldRegSlave_to_MT101 := "dbHoldRegSlave_to_MT101".instMinutStopt_Filling,
                           memRisingTriger_Data_ := "memRisingTriger_Data_8",
                           "dbHold_RRG.Sending" := "dbHold_RRG".SendingTimes.Stop_napełnianie.MINUTE,
                           ENO => #_w1);
   IF #_w1 THEN
       "08_C_Saving_Changed_Data_Word_USint"(dbHpld_RRG_set := "dbHold_RRG".Stop_napełnianie.MINUTE,
                               dbHoldRegSlave_MT101_inst := "dbHoldRegSlave_to_MT101".instMinutStopt_Filling,
                               memTrig_Client_Receiving := "memTrig_Client_Receiving_8");
   END_IF;
END_REGION

REGION Network 10: Start przetłaczanie (miasto) godzina
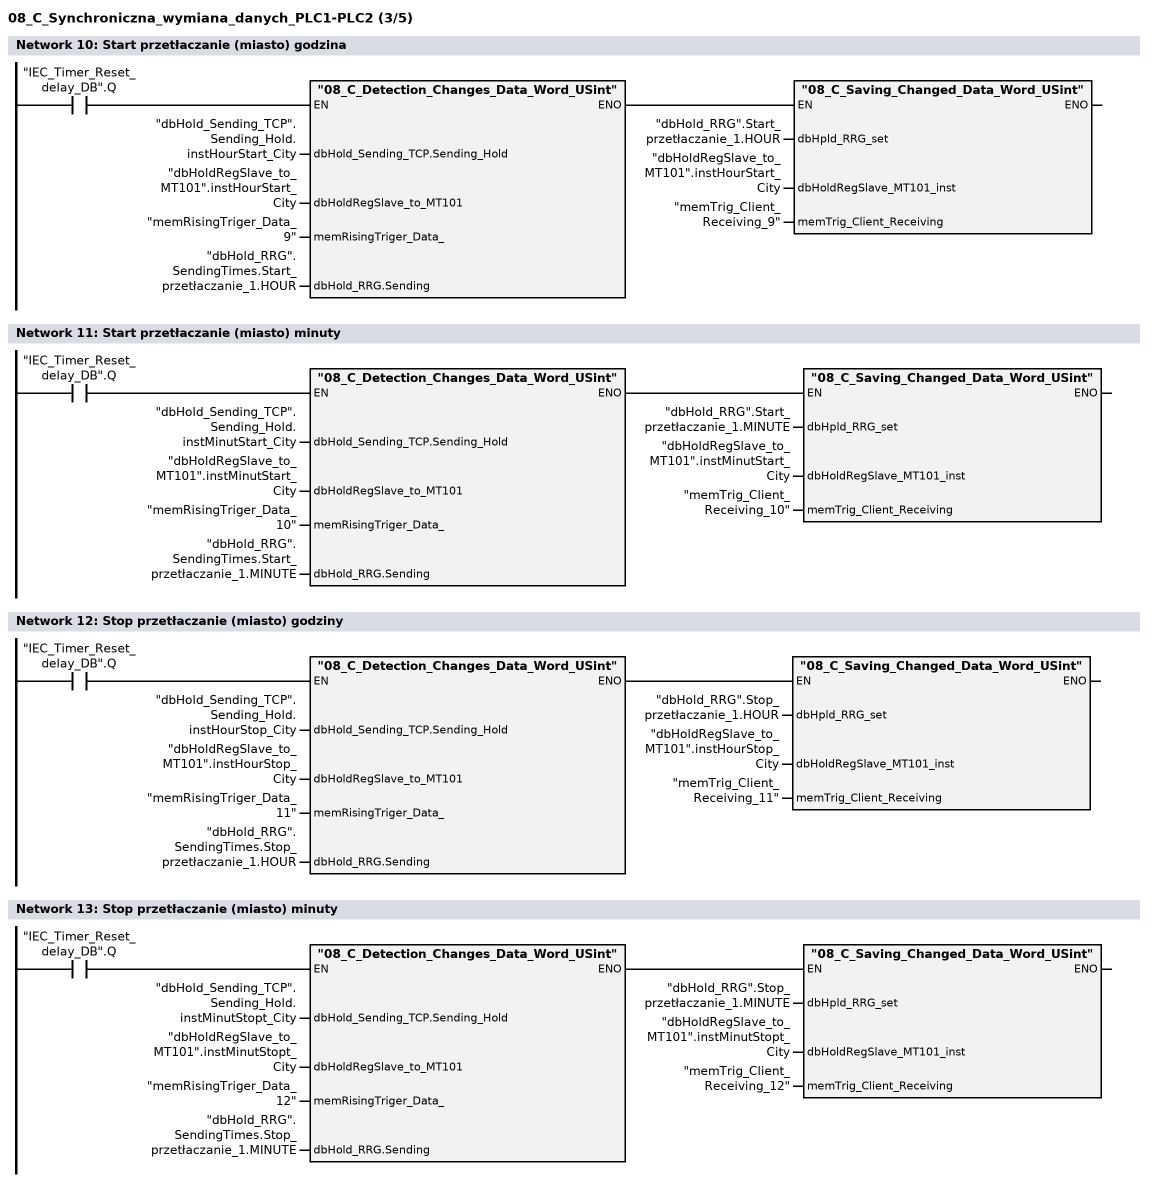
   RUNG wire#powerrail
      Contact( "IEC_Timer_Reset_delay_DB".Q )
      "08_C_Detection_Changes_Data_Word_USint"("dbHold_Sending_TCP.Sending_Hold" := "dbHold_Sending_TCP".Sending_Hold.instHourStart_City, dbHoldRegSlave_to_MT101 := "dbHoldRegSlave_to_MT101".instHourStart_City, memRisingTriger_Data_ := "memRisingTriger_Data_9", "dbHold_RRG.Sending" := "dbHold_RRG".SendingTimes.Start_przetłaczanie_1.HOUR)
      "08_C_Saving_Changed_Data_Word_USint"(dbHpld_RRG_set := "dbHold_RRG".Start_przetłaczanie_1.HOUR, dbHoldRegSlave_MT101_inst := "dbHoldRegSlave_to_MT101".instHourStart_City, memTrig_Client_Receiving := "memTrig_Client_Receiving_9")
   END_RUNG
   // the same network as SCL:
   "08_C_Detection_Changes_Data_Word_USint"(EN := "IEC_Timer_Reset_delay_DB".Q,
                           "dbHold_Sending_TCP.Sending_Hold" := "dbHold_Sending_TCP".Sending_Hold.instHourStart_City,
                           dbHoldRegSlave_to_MT101 := "dbHoldRegSlave_to_MT101".instHourStart_City,
                           memRisingTriger_Data_ := "memRisingTriger_Data_9",
                           "dbHold_RRG.Sending" := "dbHold_RRG".SendingTimes.Start_przetłaczanie_1.HOUR,
                           ENO => #_w1);
   IF #_w1 THEN
       "08_C_Saving_Changed_Data_Word_USint"(dbHpld_RRG_set := "dbHold_RRG".Start_przetłaczanie_1.HOUR,
                               dbHoldRegSlave_MT101_inst := "dbHoldRegSlave_to_MT101".instHourStart_City,
                               memTrig_Client_Receiving := "memTrig_Client_Receiving_9");
   END_IF;
END_REGION

REGION Network 11: Start przetłaczanie (miasto) minuty
   RUNG wire#powerrail
      Contact( "IEC_Timer_Reset_delay_DB".Q )
      "08_C_Detection_Changes_Data_Word_USint"("dbHold_Sending_TCP.Sending_Hold" := "dbHold_Sending_TCP".Sending_Hold.instMinutStart_City, dbHoldRegSlave_to_MT101 := "dbHoldRegSlave_to_MT101".instMinutStart_City, memRisingTriger_Data_ := "memRisingTriger_Data_10", "dbHold_RRG.Sending" := "dbHold_RRG".SendingTimes.Start_przetłaczanie_1.MINUTE)
      "08_C_Saving_Changed_Data_Word_USint"(dbHpld_RRG_set := "dbHold_RRG".Start_przetłaczanie_1.MINUTE, dbHoldRegSlave_MT101_inst := "dbHoldRegSlave_to_MT101".instMinutStart_City, memTrig_Client_Receiving := "memTrig_Client_Receiving_10")
   END_RUNG
   // the same network as SCL:
   "08_C_Detection_Changes_Data_Word_USint"(EN := "IEC_Timer_Reset_delay_DB".Q,
                           "dbHold_Sending_TCP.Sending_Hold" := "dbHold_Sending_TCP".Sending_Hold.instMinutStart_City,
                           dbHoldRegSlave_to_MT101 := "dbHoldRegSlave_to_MT101".instMinutStart_City,
                           memRisingTriger_Data_ := "memRisingTriger_Data_10",
                           "dbHold_RRG.Sending" := "dbHold_RRG".SendingTimes.Start_przetłaczanie_1.MINUTE,
                           ENO => #_w1);
   IF #_w1 THEN
       "08_C_Saving_Changed_Data_Word_USint"(dbHpld_RRG_set := "dbHold_RRG".Start_przetłaczanie_1.MINUTE,
                               dbHoldRegSlave_MT101_inst := "dbHoldRegSlave_to_MT101".instMinutStart_City,
                               memTrig_Client_Receiving := "memTrig_Client_Receiving_10");
   END_IF;
END_REGION

REGION Network 12: Stop przetłaczanie (miasto) godziny
   RUNG wire#powerrail
      Contact( "IEC_Timer_Reset_delay_DB".Q )
      "08_C_Detection_Changes_Data_Word_USint"("dbHold_Sending_TCP.Sending_Hold" := "dbHold_Sending_TCP".Sending_Hold.instHourStop_City, dbHoldRegSlave_to_MT101 := "dbHoldRegSlave_to_MT101".instHourStop_City, memRisingTriger_Data_ := "memRisingTriger_Data_11", "dbHold_RRG.Sending" := "dbHold_RRG".SendingTimes.Stop_przetłaczanie_1.HOUR)
      "08_C_Saving_Changed_Data_Word_USint"(dbHpld_RRG_set := "dbHold_RRG".Stop_przetłaczanie_1.HOUR, dbHoldRegSlave_MT101_inst := "dbHoldRegSlave_to_MT101".instHourStop_City, memTrig_Client_Receiving := "memTrig_Client_Receiving_11")
   END_RUNG
   // the same network as SCL:
   "08_C_Detection_Changes_Data_Word_USint"(EN := "IEC_Timer_Reset_delay_DB".Q,
                           "dbHold_Sending_TCP.Sending_Hold" := "dbHold_Sending_TCP".Sending_Hold.instHourStop_City,
                           dbHoldRegSlave_to_MT101 := "dbHoldRegSlave_to_MT101".instHourStop_City,
                           memRisingTriger_Data_ := "memRisingTriger_Data_11",
                           "dbHold_RRG.Sending" := "dbHold_RRG".SendingTimes.Stop_przetłaczanie_1.HOUR,
                           ENO => #_w1);
   IF #_w1 THEN
       "08_C_Saving_Changed_Data_Word_USint"(dbHpld_RRG_set := "dbHold_RRG".Stop_przetłaczanie_1.HOUR,
                               dbHoldRegSlave_MT101_inst := "dbHoldRegSlave_to_MT101".instHourStop_City,
                               memTrig_Client_Receiving := "memTrig_Client_Receiving_11");
   END_IF;
END_REGION

REGION Network 13: Stop przetłaczanie (miasto) minuty
   RUNG wire#powerrail
      Contact( "IEC_Timer_Reset_delay_DB".Q )
      "08_C_Detection_Changes_Data_Word_USint"("dbHold_Sending_TCP.Sending_Hold" := "dbHold_Sending_TCP".Sending_Hold.instMinutStopt_City, dbHoldRegSlave_to_MT101 := "dbHoldRegSlave_to_MT101".instMinutStopt_City, memRisingTriger_Data_ := "memRisingTriger_Data_12", "dbHold_RRG.Sending" := "dbHold_RRG".SendingTimes.Stop_przetłaczanie_1.MINUTE)
      "08_C_Saving_Changed_Data_Word_USint"(dbHpld_RRG_set := "dbHold_RRG".Stop_przetłaczanie_1.MINUTE, dbHoldRegSlave_MT101_inst := "dbHoldRegSlave_to_MT101".instMinutStopt_City, memTrig_Client_Receiving := "memTrig_Client_Receiving_12")
   END_RUNG
   // the same network as SCL:
   "08_C_Detection_Changes_Data_Word_USint"(EN := "IEC_Timer_Reset_delay_DB".Q,
                           "dbHold_Sending_TCP.Sending_Hold" := "dbHold_Sending_TCP".Sending_Hold.instMinutStopt_City,
                           dbHoldRegSlave_to_MT101 := "dbHoldRegSlave_to_MT101".instMinutStopt_City,
                           memRisingTriger_Data_ := "memRisingTriger_Data_12",
                           "dbHold_RRG.Sending" := "dbHold_RRG".SendingTimes.Stop_przetłaczanie_1.MINUTE,
                           ENO => #_w1);
   IF #_w1 THEN
       "08_C_Saving_Changed_Data_Word_USint"(dbHpld_RRG_set := "dbHold_RRG".Stop_przetłaczanie_1.MINUTE,
                               dbHoldRegSlave_MT101_inst := "dbHoldRegSlave_to_MT101".instMinutStopt_City,
                               memTrig_Client_Receiving := "memTrig_Client_Receiving_12");
   END_IF;
END_REGION

REGION Network 14: Start dosilanie godziny
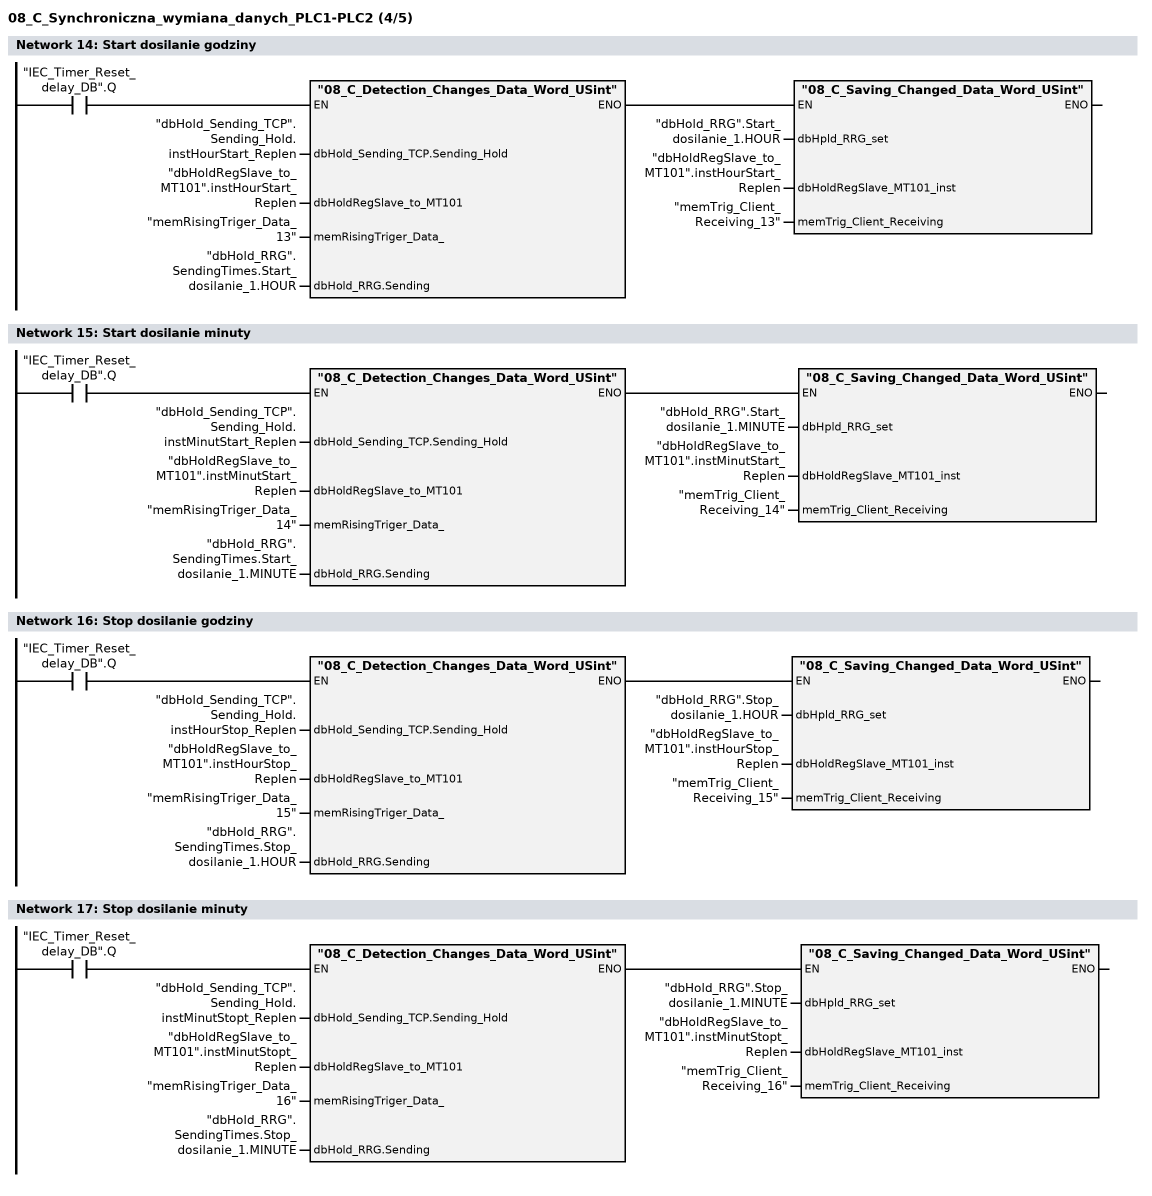
   RUNG wire#powerrail
      Contact( "IEC_Timer_Reset_delay_DB".Q )
      "08_C_Detection_Changes_Data_Word_USint"("dbHold_Sending_TCP.Sending_Hold" := "dbHold_Sending_TCP".Sending_Hold.instHourStart_Replen, dbHoldRegSlave_to_MT101 := "dbHoldRegSlave_to_MT101".instHourStart_Replen, memRisingTriger_Data_ := "memRisingTriger_Data_13", "dbHold_RRG.Sending" := "dbHold_RRG".SendingTimes.Start_dosilanie_1.HOUR)
      "08_C_Saving_Changed_Data_Word_USint"(dbHpld_RRG_set := "dbHold_RRG".Start_dosilanie_1.HOUR, dbHoldRegSlave_MT101_inst := "dbHoldRegSlave_to_MT101".instHourStart_Replen, memTrig_Client_Receiving := "memTrig_Client_Receiving_13")
   END_RUNG
   // the same network as SCL:
   "08_C_Detection_Changes_Data_Word_USint"(EN := "IEC_Timer_Reset_delay_DB".Q,
                           "dbHold_Sending_TCP.Sending_Hold" := "dbHold_Sending_TCP".Sending_Hold.instHourStart_Replen,
                           dbHoldRegSlave_to_MT101 := "dbHoldRegSlave_to_MT101".instHourStart_Replen,
                           memRisingTriger_Data_ := "memRisingTriger_Data_13",
                           "dbHold_RRG.Sending" := "dbHold_RRG".SendingTimes.Start_dosilanie_1.HOUR,
                           ENO => #_w1);
   IF #_w1 THEN
       "08_C_Saving_Changed_Data_Word_USint"(dbHpld_RRG_set := "dbHold_RRG".Start_dosilanie_1.HOUR,
                               dbHoldRegSlave_MT101_inst := "dbHoldRegSlave_to_MT101".instHourStart_Replen,
                               memTrig_Client_Receiving := "memTrig_Client_Receiving_13");
   END_IF;
END_REGION

REGION Network 15: Start dosilanie minuty
   RUNG wire#powerrail
      Contact( "IEC_Timer_Reset_delay_DB".Q )
      "08_C_Detection_Changes_Data_Word_USint"("dbHold_Sending_TCP.Sending_Hold" := "dbHold_Sending_TCP".Sending_Hold.instMinutStart_Replen, dbHoldRegSlave_to_MT101 := "dbHoldRegSlave_to_MT101".instMinutStart_Replen, memRisingTriger_Data_ := "memRisingTriger_Data_14", "dbHold_RRG.Sending" := "dbHold_RRG".SendingTimes.Start_dosilanie_1.MINUTE)
      "08_C_Saving_Changed_Data_Word_USint"(dbHpld_RRG_set := "dbHold_RRG".Start_dosilanie_1.MINUTE, dbHoldRegSlave_MT101_inst := "dbHoldRegSlave_to_MT101".instMinutStart_Replen, memTrig_Client_Receiving := "memTrig_Client_Receiving_14")
   END_RUNG
   // the same network as SCL:
   "08_C_Detection_Changes_Data_Word_USint"(EN := "IEC_Timer_Reset_delay_DB".Q,
                           "dbHold_Sending_TCP.Sending_Hold" := "dbHold_Sending_TCP".Sending_Hold.instMinutStart_Replen,
                           dbHoldRegSlave_to_MT101 := "dbHoldRegSlave_to_MT101".instMinutStart_Replen,
                           memRisingTriger_Data_ := "memRisingTriger_Data_14",
                           "dbHold_RRG.Sending" := "dbHold_RRG".SendingTimes.Start_dosilanie_1.MINUTE,
                           ENO => #_w1);
   IF #_w1 THEN
       "08_C_Saving_Changed_Data_Word_USint"(dbHpld_RRG_set := "dbHold_RRG".Start_dosilanie_1.MINUTE,
                               dbHoldRegSlave_MT101_inst := "dbHoldRegSlave_to_MT101".instMinutStart_Replen,
                               memTrig_Client_Receiving := "memTrig_Client_Receiving_14");
   END_IF;
END_REGION

REGION Network 16: Stop dosilanie godziny
   RUNG wire#powerrail
      Contact( "IEC_Timer_Reset_delay_DB".Q )
      "08_C_Detection_Changes_Data_Word_USint"("dbHold_Sending_TCP.Sending_Hold" := "dbHold_Sending_TCP".Sending_Hold.instHourStop_Replen, dbHoldRegSlave_to_MT101 := "dbHoldRegSlave_to_MT101".instHourStop_Replen, memRisingTriger_Data_ := "memRisingTriger_Data_15", "dbHold_RRG.Sending" := "dbHold_RRG".SendingTimes.Stop_dosilanie_1.HOUR)
      "08_C_Saving_Changed_Data_Word_USint"(dbHpld_RRG_set := "dbHold_RRG".Stop_dosilanie_1.HOUR, dbHoldRegSlave_MT101_inst := "dbHoldRegSlave_to_MT101".instHourStop_Replen, memTrig_Client_Receiving := "memTrig_Client_Receiving_15")
   END_RUNG
   // the same network as SCL:
   "08_C_Detection_Changes_Data_Word_USint"(EN := "IEC_Timer_Reset_delay_DB".Q,
                           "dbHold_Sending_TCP.Sending_Hold" := "dbHold_Sending_TCP".Sending_Hold.instHourStop_Replen,
                           dbHoldRegSlave_to_MT101 := "dbHoldRegSlave_to_MT101".instHourStop_Replen,
                           memRisingTriger_Data_ := "memRisingTriger_Data_15",
                           "dbHold_RRG.Sending" := "dbHold_RRG".SendingTimes.Stop_dosilanie_1.HOUR,
                           ENO => #_w1);
   IF #_w1 THEN
       "08_C_Saving_Changed_Data_Word_USint"(dbHpld_RRG_set := "dbHold_RRG".Stop_dosilanie_1.HOUR,
                               dbHoldRegSlave_MT101_inst := "dbHoldRegSlave_to_MT101".instHourStop_Replen,
                               memTrig_Client_Receiving := "memTrig_Client_Receiving_15");
   END_IF;
END_REGION

REGION Network 17: Stop dosilanie minuty
   RUNG wire#powerrail
      Contact( "IEC_Timer_Reset_delay_DB".Q )
      "08_C_Detection_Changes_Data_Word_USint"("dbHold_Sending_TCP.Sending_Hold" := "dbHold_Sending_TCP".Sending_Hold.instMinutStopt_Replen, dbHoldRegSlave_to_MT101 := "dbHoldRegSlave_to_MT101".instMinutStopt_Replen, memRisingTriger_Data_ := "memRisingTriger_Data_16", "dbHold_RRG.Sending" := "dbHold_RRG".SendingTimes.Stop_dosilanie_1.MINUTE)
      "08_C_Saving_Changed_Data_Word_USint"(dbHpld_RRG_set := "dbHold_RRG".Stop_dosilanie_1.MINUTE, dbHoldRegSlave_MT101_inst := "dbHoldRegSlave_to_MT101".instMinutStopt_Replen, memTrig_Client_Receiving := "memTrig_Client_Receiving_16")
   END_RUNG
   // the same network as SCL:
   "08_C_Detection_Changes_Data_Word_USint"(EN := "IEC_Timer_Reset_delay_DB".Q,
                           "dbHold_Sending_TCP.Sending_Hold" := "dbHold_Sending_TCP".Sending_Hold.instMinutStopt_Replen,
                           dbHoldRegSlave_to_MT101 := "dbHoldRegSlave_to_MT101".instMinutStopt_Replen,
                           memRisingTriger_Data_ := "memRisingTriger_Data_16",
                           "dbHold_RRG.Sending" := "dbHold_RRG".SendingTimes.Stop_dosilanie_1.MINUTE,
                           ENO => #_w1);
   IF #_w1 THEN
       "08_C_Saving_Changed_Data_Word_USint"(dbHpld_RRG_set := "dbHold_RRG".Stop_dosilanie_1.MINUTE,
                               dbHoldRegSlave_MT101_inst := "dbHoldRegSlave_to_MT101".instMinutStopt_Replen,
                               memTrig_Client_Receiving := "memTrig_Client_Receiving_16");
   END_IF;
END_REGION

REGION Network 19: Wybór trymu pracy M1,M2,M3,M4, Z1-Z8
   // dbHoldRegSlave_MT101 - tu wartość zadajemy 
   // dbHoldSending_TCP.Sending_Hold - z tą wzmienną porównujemy 
   // dbHold_REG.Sending - tu wysyłamy
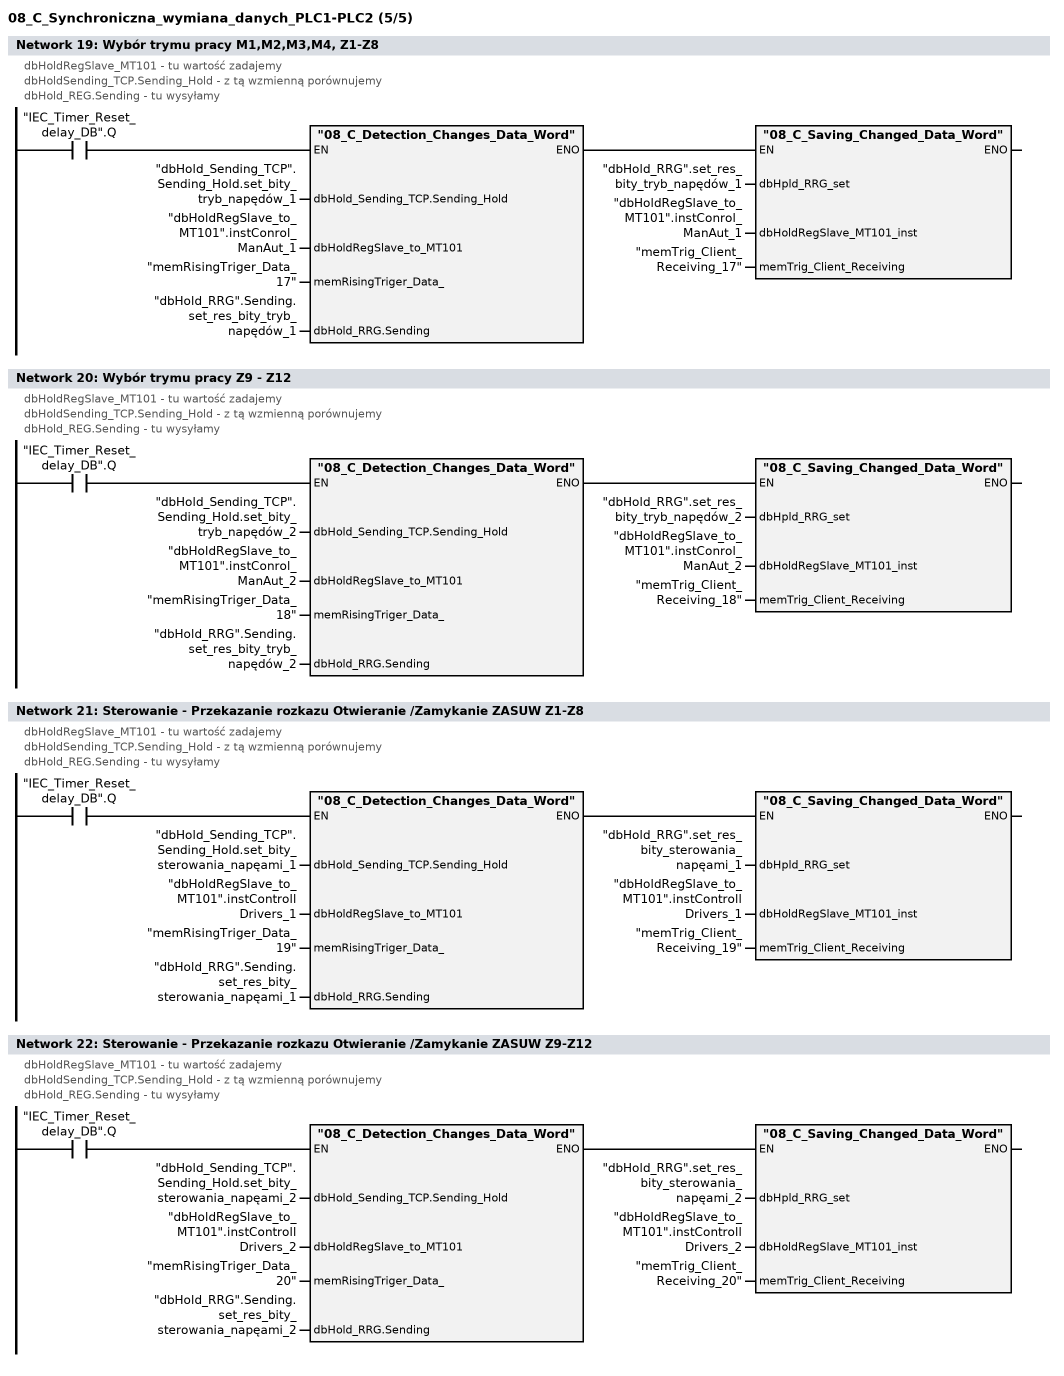
   RUNG wire#powerrail
      Contact( "IEC_Timer_Reset_delay_DB".Q )
      "08_C_Detection_Changes_Data_Word"("dbHold_Sending_TCP.Sending_Hold" := "dbHold_Sending_TCP".Sending_Hold.set_bity_tryb_napędów_1, dbHoldRegSlave_to_MT101 := "dbHoldRegSlave_to_MT101".instConrol_ManAut_1, memRisingTriger_Data_ := "memRisingTriger_Data_17", "dbHold_RRG.Sending" := "dbHold_RRG".Sending.set_res_bity_tryb_napędów_1)
      "08_C_Saving_Changed_Data_Word"(dbHpld_RRG_set := "dbHold_RRG".set_res_bity_tryb_napędów_1, dbHoldRegSlave_MT101_inst := "dbHoldRegSlave_to_MT101".instConrol_ManAut_1, memTrig_Client_Receiving := "memTrig_Client_Receiving_17")
   END_RUNG
   // the same network as SCL:
   "08_C_Detection_Changes_Data_Word"(EN := "IEC_Timer_Reset_delay_DB".Q,
                           "dbHold_Sending_TCP.Sending_Hold" := "dbHold_Sending_TCP".Sending_Hold.set_bity_tryb_napędów_1,
                           dbHoldRegSlave_to_MT101 := "dbHoldRegSlave_to_MT101".instConrol_ManAut_1,
                           memRisingTriger_Data_ := "memRisingTriger_Data_17",
                           "dbHold_RRG.Sending" := "dbHold_RRG".Sending.set_res_bity_tryb_napędów_1,
                           ENO => #_w1);
   IF #_w1 THEN
       "08_C_Saving_Changed_Data_Word"(dbHpld_RRG_set := "dbHold_RRG".set_res_bity_tryb_napędów_1,
                               dbHoldRegSlave_MT101_inst := "dbHoldRegSlave_to_MT101".instConrol_ManAut_1,
                               memTrig_Client_Receiving := "memTrig_Client_Receiving_17");
   END_IF;
END_REGION

REGION Network 20: Wybór trymu pracy Z9 - Z12
   // dbHoldRegSlave_MT101 - tu wartość zadajemy 
   // dbHoldSending_TCP.Sending_Hold - z tą wzmienną porównujemy 
   // dbHold_REG.Sending - tu wysyłamy
   RUNG wire#powerrail
      Contact( "IEC_Timer_Reset_delay_DB".Q )
      "08_C_Detection_Changes_Data_Word"("dbHold_Sending_TCP.Sending_Hold" := "dbHold_Sending_TCP".Sending_Hold.set_bity_tryb_napędów_2, dbHoldRegSlave_to_MT101 := "dbHoldRegSlave_to_MT101".instConrol_ManAut_2, memRisingTriger_Data_ := "memRisingTriger_Data_18", "dbHold_RRG.Sending" := "dbHold_RRG".Sending.set_res_bity_tryb_napędów_2)
      "08_C_Saving_Changed_Data_Word"(dbHpld_RRG_set := "dbHold_RRG".set_res_bity_tryb_napędów_2, dbHoldRegSlave_MT101_inst := "dbHoldRegSlave_to_MT101".instConrol_ManAut_2, memTrig_Client_Receiving := "memTrig_Client_Receiving_18")
   END_RUNG
   // the same network as SCL:
   "08_C_Detection_Changes_Data_Word"(EN := "IEC_Timer_Reset_delay_DB".Q,
                           "dbHold_Sending_TCP.Sending_Hold" := "dbHold_Sending_TCP".Sending_Hold.set_bity_tryb_napędów_2,
                           dbHoldRegSlave_to_MT101 := "dbHoldRegSlave_to_MT101".instConrol_ManAut_2,
                           memRisingTriger_Data_ := "memRisingTriger_Data_18",
                           "dbHold_RRG.Sending" := "dbHold_RRG".Sending.set_res_bity_tryb_napędów_2,
                           ENO => #_w1);
   IF #_w1 THEN
       "08_C_Saving_Changed_Data_Word"(dbHpld_RRG_set := "dbHold_RRG".set_res_bity_tryb_napędów_2,
                               dbHoldRegSlave_MT101_inst := "dbHoldRegSlave_to_MT101".instConrol_ManAut_2,
                               memTrig_Client_Receiving := "memTrig_Client_Receiving_18");
   END_IF;
END_REGION

REGION Network 21: Sterowanie - Przekazanie rozkazu Otwieranie /Zamykanie ZASUW Z1-Z8
   // dbHoldRegSlave_MT101 - tu wartość zadajemy 
   // dbHoldSending_TCP.Sending_Hold - z tą wzmienną porównujemy 
   // dbHold_REG.Sending - tu wysyłamy
   RUNG wire#powerrail
      Contact( "IEC_Timer_Reset_delay_DB".Q )
      "08_C_Detection_Changes_Data_Word"("dbHold_Sending_TCP.Sending_Hold" := "dbHold_Sending_TCP".Sending_Hold.set_bity_sterowania_napęami_1, dbHoldRegSlave_to_MT101 := "dbHoldRegSlave_to_MT101".instControllDrivers_1, memRisingTriger_Data_ := "memRisingTriger_Data_19", "dbHold_RRG.Sending" := "dbHold_RRG".Sending.set_res_bity_sterowania_napęami_1)
      "08_C_Saving_Changed_Data_Word"(dbHpld_RRG_set := "dbHold_RRG".set_res_bity_sterowania_napęami_1, dbHoldRegSlave_MT101_inst := "dbHoldRegSlave_to_MT101".instControllDrivers_1, memTrig_Client_Receiving := "memTrig_Client_Receiving_19")
   END_RUNG
   // the same network as SCL:
   "08_C_Detection_Changes_Data_Word"(EN := "IEC_Timer_Reset_delay_DB".Q,
                           "dbHold_Sending_TCP.Sending_Hold" := "dbHold_Sending_TCP".Sending_Hold.set_bity_sterowania_napęami_1,
                           dbHoldRegSlave_to_MT101 := "dbHoldRegSlave_to_MT101".instControllDrivers_1,
                           memRisingTriger_Data_ := "memRisingTriger_Data_19",
                           "dbHold_RRG.Sending" := "dbHold_RRG".Sending.set_res_bity_sterowania_napęami_1,
                           ENO => #_w1);
   IF #_w1 THEN
       "08_C_Saving_Changed_Data_Word"(dbHpld_RRG_set := "dbHold_RRG".set_res_bity_sterowania_napęami_1,
                               dbHoldRegSlave_MT101_inst := "dbHoldRegSlave_to_MT101".instControllDrivers_1,
                               memTrig_Client_Receiving := "memTrig_Client_Receiving_19");
   END_IF;
END_REGION

REGION Network 22: Sterowanie - Przekazanie rozkazu Otwieranie /Zamykanie ZASUW Z9-Z12
   // dbHoldRegSlave_MT101 - tu wartość zadajemy 
   // dbHoldSending_TCP.Sending_Hold - z tą wzmienną porównujemy 
   // dbHold_REG.Sending - tu wysyłamy
   RUNG wire#powerrail
      Contact( "IEC_Timer_Reset_delay_DB".Q )
      "08_C_Detection_Changes_Data_Word"("dbHold_Sending_TCP.Sending_Hold" := "dbHold_Sending_TCP".Sending_Hold.set_bity_sterowania_napęami_2, dbHoldRegSlave_to_MT101 := "dbHoldRegSlave_to_MT101".instControllDrivers_2, memRisingTriger_Data_ := "memRisingTriger_Data_20", "dbHold_RRG.Sending" := "dbHold_RRG".Sending.set_res_bity_sterowania_napęami_2)
      "08_C_Saving_Changed_Data_Word"(dbHpld_RRG_set := "dbHold_RRG".set_res_bity_sterowania_napęami_2, dbHoldRegSlave_MT101_inst := "dbHoldRegSlave_to_MT101".instControllDrivers_2, memTrig_Client_Receiving := "memTrig_Client_Receiving_20")
   END_RUNG
   // the same network as SCL:
   "08_C_Detection_Changes_Data_Word"(EN := "IEC_Timer_Reset_delay_DB".Q,
                           "dbHold_Sending_TCP.Sending_Hold" := "dbHold_Sending_TCP".Sending_Hold.set_bity_sterowania_napęami_2,
                           dbHoldRegSlave_to_MT101 := "dbHoldRegSlave_to_MT101".instControllDrivers_2,
                           memRisingTriger_Data_ := "memRisingTriger_Data_20",
                           "dbHold_RRG.Sending" := "dbHold_RRG".Sending.set_res_bity_sterowania_napęami_2,
                           ENO => #_w1);
   IF #_w1 THEN
       "08_C_Saving_Changed_Data_Word"(dbHpld_RRG_set := "dbHold_RRG".set_res_bity_sterowania_napęami_2,
                               dbHoldRegSlave_MT101_inst := "dbHoldRegSlave_to_MT101".instControllDrivers_2,
                               memTrig_Client_Receiving := "memTrig_Client_Receiving_20");
   END_IF;
END_REGION
END_FUNCTION

FUNCTION "08_C_Detection_Changes_Data_Real" : Void   // FC60, LAD
{ S7_Optimized_Access := 'TRUE' }
AUTHOR : rtecmer
VERSION : 0.1
// stored: AutoNumber true, IsIECCheckEnabled false, SetENOAutomatically false, UDAEnableTagReadback false
   VAR_IN_OUT
      "dbHold_Sending_TCP.Sending_Hold" : Real;   // Zmienna zadająca i porównywana
      dbHoldRegSlave_to_MT101 : Real;   // Zmienna w db do której porównujemy
      memRisingTriger_Data_ : Bool;   // bit pamięć zmiany
      "dbHold_RRG.Sending" : Real;   // zmienna docelowa w db do wysłania
   END_VAR
   VAR_TEMP   // added for the SCL form of the ladder/FBD networks
      _w1 : Bool;
      _w2 : Bool;
   END_VAR
BEGIN

REGION Network 1: set_poziom_napełniania
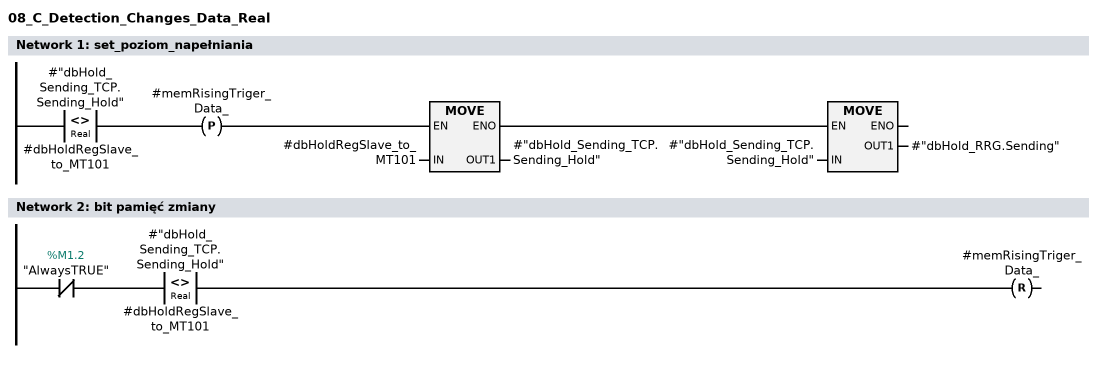
   RUNG wire#powerrail
      { S7_Templates := "SrcType := Real" } NE_Contact(in1 := #"dbHold_Sending_TCP.Sending_Hold", in2 := #dbHoldRegSlave_to_MT101)
      P_Trig( #memRisingTriger_Data_ )
      Move(in := #dbHoldRegSlave_to_MT101, out1 => #"dbHold_Sending_TCP.Sending_Hold")
      Move(in := #"dbHold_Sending_TCP.Sending_Hold", out1 => #"dbHold_RRG.Sending")
   END_RUNG
   // the same network as SCL:
   #_w1 := #"dbHold_Sending_TCP.Sending_Hold" <> #dbHoldRegSlave_to_MT101;
   #_w2 := #_w1 AND NOT #memRisingTriger_Data_;   // rising edge
   #memRisingTriger_Data_ := #_w1;
   IF #_w2 THEN
       #"dbHold_Sending_TCP.Sending_Hold" := #dbHoldRegSlave_to_MT101;
       #"dbHold_RRG.Sending" := #"dbHold_Sending_TCP.Sending_Hold";
   END_IF;
END_REGION

REGION Network 2: bit pamięć zmiany
   RUNG wire#powerrail
      I_Contact( "AlwaysTRUE" )
      { S7_Templates := "SrcType := Real" } NE_Contact(in1 := #"dbHold_Sending_TCP.Sending_Hold", in2 := #dbHoldRegSlave_to_MT101)
      R_Coil( #memRisingTriger_Data_ )
   END_RUNG
   // the same network as SCL:
   IF NOT "AlwaysTRUE" AND (#"dbHold_Sending_TCP.Sending_Hold" <> #dbHoldRegSlave_to_MT101) THEN
       #memRisingTriger_Data_ := FALSE;
   END_IF;
END_REGION
END_FUNCTION

FUNCTION "08_C_Saving_Changed_Data_Real" : Void   // FC58, LAD
{ S7_Optimized_Access := 'TRUE' }
AUTHOR : rtecmer
VERSION : 0.1
// Porównanie czy doszło do zmiany watości w db Hold_RRG <> db HoldRegSlave_toMT101
// stored: AutoNumber true, IsIECCheckEnabled false, SetENOAutomatically false, UDAEnableTagReadback false
   VAR_IN_OUT
      dbHpld_RRG_set : Real;   // Wartość zadawana porównywana
      dbHoldRegSlave_MT101_inst : Real;   // Wartość do której porównujemy
      memTrig_Client_Receiving : Bool;   // pamiec zbocza zmiany
   END_VAR
   VAR_TEMP   // added for the SCL form of the ladder/FBD networks
      _w1 : Bool;
      _w2 : Bool;
   END_VAR
BEGIN

REGION Network 1
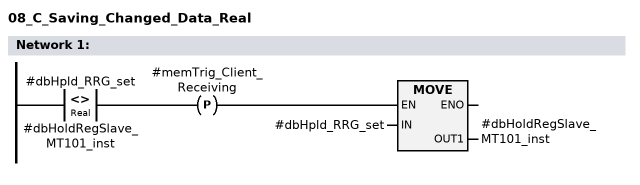
   RUNG wire#powerrail
      { S7_Templates := "SrcType := Real" } NE_Contact(in1 := #dbHpld_RRG_set, in2 := #dbHoldRegSlave_MT101_inst)
      P_Trig( #memTrig_Client_Receiving )
      Move(in := #dbHpld_RRG_set, out1 => #dbHoldRegSlave_MT101_inst)
   END_RUNG
   // the same network as SCL:
   #_w1 := #dbHpld_RRG_set <> #dbHoldRegSlave_MT101_inst;
   #_w2 := #_w1 AND NOT #memTrig_Client_Receiving;   // rising edge
   #memTrig_Client_Receiving := #_w1;
   IF #_w2 THEN #dbHoldRegSlave_MT101_inst := #dbHpld_RRG_set; END_IF;
END_REGION
END_FUNCTION

FUNCTION "08_C_Detection_Changes_Data_Word" : Void   // FC62, LAD
{ S7_Optimized_Access := 'TRUE' }
AUTHOR : rtecmer
VERSION : 0.1
// stored: AutoNumber false, IsIECCheckEnabled false, SetENOAutomatically false, UDAEnableTagReadback false
   VAR_IN_OUT
      "dbHold_Sending_TCP.Sending_Hold" : Int;   // Zmienna zadająca i porównywana
      dbHoldRegSlave_to_MT101 : Int;   // Zmienna w db do której porównujemy
      memRisingTriger_Data_ : Bool;   // bit pamięć zmiany
      "dbHold_RRG.Sending" : Int;   // zmienna docelowa w db do wysłania
   END_VAR
   VAR_TEMP   // added for the SCL form of the ladder/FBD networks
      _w1 : Bool;
      _w2 : Bool;
   END_VAR
BEGIN

REGION Network 1: set_poziom_napełniania
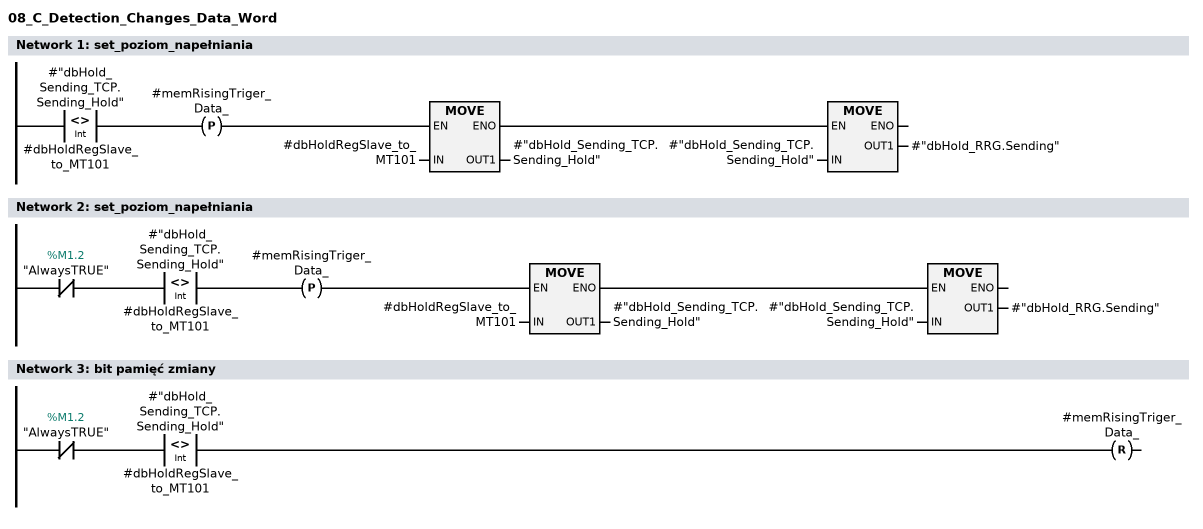
   RUNG wire#powerrail
      { S7_Templates := "SrcType := Int" } NE_Contact(in1 := #"dbHold_Sending_TCP.Sending_Hold", in2 := #dbHoldRegSlave_to_MT101)
      P_Trig( #memRisingTriger_Data_ )
      Move(in := #dbHoldRegSlave_to_MT101, out1 => #"dbHold_Sending_TCP.Sending_Hold")
      Move(in := #"dbHold_Sending_TCP.Sending_Hold", out1 => #"dbHold_RRG.Sending")
   END_RUNG
   // the same network as SCL:
   #_w1 := #"dbHold_Sending_TCP.Sending_Hold" <> #dbHoldRegSlave_to_MT101;
   #_w2 := #_w1 AND NOT #memRisingTriger_Data_;   // rising edge
   #memRisingTriger_Data_ := #_w1;
   IF #_w2 THEN
       #"dbHold_Sending_TCP.Sending_Hold" := #dbHoldRegSlave_to_MT101;
       #"dbHold_RRG.Sending" := #"dbHold_Sending_TCP.Sending_Hold";
   END_IF;
END_REGION

REGION Network 2: set_poziom_napełniania
   RUNG wire#powerrail
      I_Contact( "AlwaysTRUE" )
      { S7_Templates := "SrcType := Int" } NE_Contact(in1 := #"dbHold_Sending_TCP.Sending_Hold", in2 := #dbHoldRegSlave_to_MT101)
      P_Trig( #memRisingTriger_Data_ )
      Move(in := #dbHoldRegSlave_to_MT101, out1 => #"dbHold_Sending_TCP.Sending_Hold")
      Move(in := #"dbHold_Sending_TCP.Sending_Hold", out1 => #"dbHold_RRG.Sending")
   END_RUNG
   // the same network as SCL:
   #_w1 := NOT "AlwaysTRUE" AND (#"dbHold_Sending_TCP.Sending_Hold" <> #dbHoldRegSlave_to_MT101);
   #_w2 := #_w1 AND NOT #memRisingTriger_Data_;   // rising edge
   #memRisingTriger_Data_ := #_w1;
   IF #_w2 THEN
       #"dbHold_Sending_TCP.Sending_Hold" := #dbHoldRegSlave_to_MT101;
       #"dbHold_RRG.Sending" := #"dbHold_Sending_TCP.Sending_Hold";
   END_IF;
END_REGION

REGION Network 3: bit pamięć zmiany
   RUNG wire#powerrail
      I_Contact( "AlwaysTRUE" )
      { S7_Templates := "SrcType := Int" } NE_Contact(in1 := #"dbHold_Sending_TCP.Sending_Hold", in2 := #dbHoldRegSlave_to_MT101)
      R_Coil( #memRisingTriger_Data_ )
   END_RUNG
   // the same network as SCL:
   IF NOT "AlwaysTRUE" AND (#"dbHold_Sending_TCP.Sending_Hold" <> #dbHoldRegSlave_to_MT101) THEN
       #memRisingTriger_Data_ := FALSE;
   END_IF;
END_REGION
END_FUNCTION

FUNCTION "08_C_Saving_Changed_Data_Word" : Void   // FC59, LAD
{ S7_Optimized_Access := 'TRUE' }
AUTHOR : rtecmer
VERSION : 0.1
// Porównanie czy doszło do zmiany watości w db Hold_RRG <> db HoldRegSlave_toMT101
// stored: AutoNumber false, IsIECCheckEnabled false, SetENOAutomatically false, UDAEnableTagReadback false
   VAR_IN_OUT
      dbHpld_RRG_set : Int;   // Wartość zadawana porównywana
      dbHoldRegSlave_MT101_inst : Int;   // Wartość do której porównujemy
      memTrig_Client_Receiving : Bool;   // pamiec zbocza zmiany
   END_VAR
   VAR_TEMP   // added for the SCL form of the ladder/FBD networks
      _w1 : Bool;
      _w2 : Bool;
   END_VAR
BEGIN

REGION Network 1
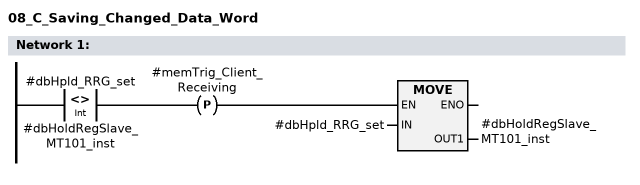
   RUNG wire#powerrail
      { S7_Templates := "SrcType := Int" } NE_Contact(in1 := #dbHpld_RRG_set, in2 := #dbHoldRegSlave_MT101_inst)
      P_Trig( #memTrig_Client_Receiving )
      Move(in := #dbHpld_RRG_set, out1 => #dbHoldRegSlave_MT101_inst)
   END_RUNG
   // the same network as SCL:
   #_w1 := #dbHpld_RRG_set <> #dbHoldRegSlave_MT101_inst;
   #_w2 := #_w1 AND NOT #memTrig_Client_Receiving;   // rising edge
   #memTrig_Client_Receiving := #_w1;
   IF #_w2 THEN #dbHoldRegSlave_MT101_inst := #dbHpld_RRG_set; END_IF;
END_REGION
END_FUNCTION

FUNCTION "08_C_Detection_Changes_Data_Word_USint" : Void   // FC64, LAD
{ S7_Optimized_Access := 'TRUE' }
AUTHOR : rtecmer
VERSION : 0.1
// stored: AutoNumber false, IsIECCheckEnabled false, SetENOAutomatically false, UDAEnableTagReadback false
   VAR_IN_OUT
      "dbHold_Sending_TCP.Sending_Hold" : Int;   // Zmienna zadająca i porównywana
      dbHoldRegSlave_to_MT101 : Int;   // Zmienna w db do której porównujemy
      memRisingTriger_Data_ : Bool;   // bit pamięć zmiany
      "dbHold_RRG.Sending" : USInt;   // zmienna docelowa w db do wysłania
   END_VAR
   VAR_TEMP   // added for the SCL form of the ladder/FBD networks
      _w1 : Bool;
      _w2 : Bool;
   END_VAR
BEGIN

REGION Network 1: set_poziom_napełniania
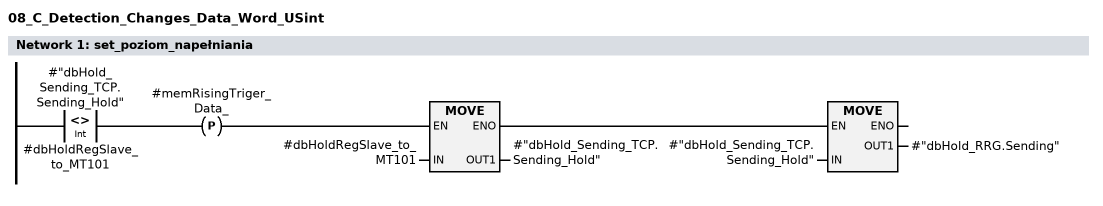
   RUNG wire#powerrail
      { S7_Templates := "SrcType := Int" } NE_Contact(in1 := #"dbHold_Sending_TCP.Sending_Hold", in2 := #dbHoldRegSlave_to_MT101)
      P_Trig( #memRisingTriger_Data_ )
      Move(in := #dbHoldRegSlave_to_MT101, out1 => #"dbHold_Sending_TCP.Sending_Hold")
      Move(in := #"dbHold_Sending_TCP.Sending_Hold", out1 => #"dbHold_RRG.Sending")
   END_RUNG
   // the same network as SCL:
   #_w1 := #"dbHold_Sending_TCP.Sending_Hold" <> #dbHoldRegSlave_to_MT101;
   #_w2 := #_w1 AND NOT #memRisingTriger_Data_;   // rising edge
   #memRisingTriger_Data_ := #_w1;
   IF #_w2 THEN
       #"dbHold_Sending_TCP.Sending_Hold" := #dbHoldRegSlave_to_MT101;
       #"dbHold_RRG.Sending" := #"dbHold_Sending_TCP.Sending_Hold";
   END_IF;
END_REGION
END_FUNCTION

FUNCTION "08_C_Saving_Changed_Data_Word_USint" : Void   // FC65, LAD
{ S7_Optimized_Access := 'TRUE' }
AUTHOR : rtecmer
VERSION : 0.1
// Porównanie czy doszło do zmiany watości w db Hold_RRG <> db HoldRegSlave_toMT101
// stored: AutoNumber false, IsIECCheckEnabled false, SetENOAutomatically false, UDAEnableTagReadback false
   VAR_IN_OUT
      dbHpld_RRG_set : USInt;   // Wartość zadawana porównywana
      dbHoldRegSlave_MT101_inst : Int;   // Wartość do której porównujemy
      memTrig_Client_Receiving : Bool;   // pamiec zbocza zmiany
   END_VAR
   VAR_TEMP   // added for the SCL form of the ladder/FBD networks
      _w1 : Bool;
      _w2 : Bool;
   END_VAR
BEGIN

REGION Network 1
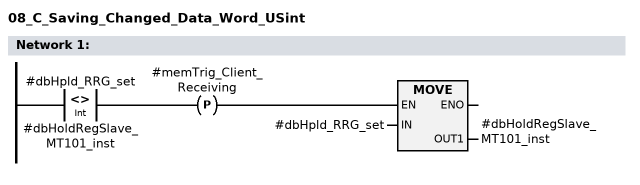
   RUNG wire#powerrail
      { S7_Templates := "SrcType := Int" } NE_Contact(in1 := #dbHpld_RRG_set, in2 := #dbHoldRegSlave_MT101_inst)
      P_Trig( #memTrig_Client_Receiving )
      Move(in := #dbHpld_RRG_set, out1 => #dbHoldRegSlave_MT101_inst)
   END_RUNG
   // the same network as SCL:
   #_w1 := #dbHpld_RRG_set <> #dbHoldRegSlave_MT101_inst;
   #_w2 := #_w1 AND NOT #memTrig_Client_Receiving;   // rising edge
   #memTrig_Client_Receiving := #_w1;
   IF #_w2 THEN #dbHoldRegSlave_MT101_inst := #dbHpld_RRG_set; END_IF;
END_REGION
END_FUNCTION

FUNCTION_BLOCK "08_C_operating_mode_select_aut-man"
TITLE = Przełącznik Trybu Pracy Napędów
{ S7_Optimized_Access := 'TRUE' }
AUTHOR : rtecmer
VERSION : 0.1
//Funkcja przeprowadza sptawdzenie stanu zmiany sygnału  na zmiennych wyboru trybu pracy napeów i jesli strwierdzi zmianę stanu zmennej to wykonuje zmianę trybu na AUT
   VAR 
      setTrig_M1 : Bool;   // bit pomocniczy przełączenia trybu
      setTrig_M2 : Bool := false;   // bit pomocniczy przełączenia trybu
      setTrig_M3 : Bool := false;   // bit pomocniczy przełączenia trybu
      setTrig_M4 : Bool := false;   // bit pomocniczy przełączenia trybu
      setTrig_Z11 : Bool := false;   // bit pomocniczy przełączenia trybu
      setTrig_Z12 : Bool := false;   // bit pomocniczy przełączenia trybu
      set_aut_man_M1 : Bool := false;   // bit pomocniczy przełączenia trybu
      set_aut_man_M2 : Bool := false;   // bit pomocniczy przełączenia trybu
      set_aut_man_M3 : Bool := false;   // bit pomocniczy przełączenia trybu
      set_aut_man_M4 : Bool := false;   // bit pomocniczy przełączenia trybu
      set_aut_man_Z11 : Bool := false;   // bit pomocniczy przełączenia trybu
      set_aut_man_Z12 : Bool := false;   // bit pomocniczy przełączenia trybu
   END_VAR


BEGIN
	(*
	//=============================================================================
	//(JZWiK S.A Radosław Tecmer)
	//(c)Copyright (2021) All Rights Reserved
	//-----------------------------------------------------------------------------
	//Testowane z:   (system docelowy z  FW 4.2)
	//Pakiet inżynierski:   TIA Portal (V14 Sp1 Update 9)
	//Ograniczenia:  ( - )
	//Wymagania:  (minimalne S7-1200 CPU 1214 FW 3.2 .)
	//Funkcjonalnośc: (Pzetwarzanie sygnałów z MT101 protokołem Modbus RTU. 
	                    Wybór Trybu Pracy Napędu)
	//-----------------------------------------------------------------------------
	//Zmainy wprowadzone:
	//Wersja  Data       Osoba wprowadzająca zmiany - ekspert
	//01.00.00 17.06.2022 (Tecmer Radosław - twórca) Pieresza wersja 01.00.00
	//=============================================================================
	*)
	
	//--- Wybór Trybu Pracy Aut/Man
	
	//Drive Motor 1 ustaw na  Automat/Manual/Start/Stop
	// Pompy
	
	REGION //Drive Motor 1 ustaw na  Automat/Manual/Start/Stop
	  // przełączniki bistabilny każdy stan Hi powoduje zmianę przełącznika
	  IF %DB100.DBX37.0 OR %DB100.DBX37.4 THEN
	    // inicjacja przełączenia
	    #set_aut_man_M1 := TRUE;
	  ELSE
	    #set_aut_man_M1 := FALSE
	    ;
	  END_IF;
	  
	  IF %DB100.DBX0.0 = FALSE THEN
	    // przełącznik bistabilny 
	    "R_TRIG_DB_AUT_M1"(CLK := #set_aut_man_M1,
	                       Q => #setTrig_M1);
	    ;
	  END_IF;
	  
	  // jeśli przełaczenie na aut
	  IF #setTrig_M1 = TRUE AND %DB100.DBX37.0 = TRUE THEN
	    %DB100.DBX0.7 := TRUE;
	    ;
	  END_IF;
	  // jeśli przełaczenie na manual
	  IF #setTrig_M1 = TRUE AND %DB100.DBX37.4 = TRUE THEN
	    %DB100.DBX0.7 := FALSE;
	    ;
	  END_IF;
	  // warunek na czyszczenie
	  IF (%DB100.DBX1.7 AND %DB100.DBX37.0) OR (%DB100.DBX1.7 = FALSE AND %DB100.DBX37.4) THEN
	    // Wyczyść całą zmienną
	    "dbHoldRegSlave_to_MT101".instConrol_ManAut_1 := 0;
	    // Kasowanie bitu 
	    %DB100.DBX37.0 := False;
	    %DB100.DBX37.4 := False;
	    ;
	  END_IF;
	  
	  // Start /
	  // przekazanie bitu roskazu z bloku modbus rtu do bloku statusu napędu
	IF %DB100.DBX33.0 THEN
	  // ustaw bit stat
	  %DB100.DBX0.5 := %DB100.DBX33.0; //ustawienie bitu start
	END_IF;
	IF %DB100.DBX33.0 AND %DB100.DBX0.3 THEN
	    //jeśli ustawiony bit startu z modbus i potwierdzone run napędu
	    %DB100.DBX33.0 := FALSE; // kasuj bit roskazu
	    ;
	  END_IF;
	  //Stop
	  // przekazanie bitu roskazu z bloku modbus rtu do bloku statusu napędu
	  IF %DB100.DBX33.4 THEN
	    %DB100.DBX0.4 := %DB100.DBX33.4;//ustawienie bitu stop
	    ;
	  END_IF;
	  IF %DB100.DBX33.4 AND %DB100.DBX0.3 = FALSE THEN
	    //jeśli ustawiony bit stop z modbus i potwierdzone stop napędu
	    %DB100.DBX33.4 := FALSE; // kasuj bit roskazu
	    ;
	  END_IF;
	  
	  
	  
	END_REGION
	
	
	REGION //Drive Motor 2 ustaw na  Automat/Manual/Stop/Start
	  // przełączniki bistabilny każdy stan Hi powoduje zmianę przełącznika
	  IF %DB100.DBX37.1 OR %DB100.DBX37.5 THEN
	    //inicjacja przełączenia
	    #set_aut_man_M2 := TRUE;
	  ELSE
	    #set_aut_man_M2 := FALSE
	    ;
	  END_IF;
	  
	  IF %DB100.DBX2.0 = FALSE THEN
	    // przełącznik bistabilny 
	    "R_TRIG_DB_AUT_M2"(CLK := #set_aut_man_M2,
	                       Q => #setTrig_M2);
	    ;
	  END_IF;
	  // pzrełącz na automat
	  IF #setTrig_M2 = TRUE AND %DB100.DBX37.1 = TRUE THEN
	    %DB100.DBX2.7 := TRUE;
	    ;
	  END_IF;
	  //przełącz na manual
	  IF #setTrig_M2 = TRUE AND %DB100.DBX37.5 = TRUE THEN
	    %DB100.DBX2.7 := FALSE;
	    ;
	  END_IF;
	  
	  IF (%DB100.DBX2.7 AND %DB100.DBX37.1) OR (%DB100.DBX2.7 = FALSE AND %DB100.DBX37.5)  THEN
	    // Wyczyść całą zmienną
	    "dbHoldRegSlave_to_MT101".instConrol_ManAut_1 := 0;
	    // Kasowanie bitu 
	    %DB100.DBX37.1 := False;
	    %DB100.DBX37.5 := FALSE;
	    ;
	  END_IF;
	  
	  // Start /
	  // przekazanie bitu roskazu z bloku modbus rtu do bloku statusu napędu
	  IF %DB100.DBX33.1 THEN // 
	    %DB100.DBX2.5 := TRUE; //ustawienie bitu start
	  END_IF;
	  IF %DB100.DBX33.1 AND %DB100.DBX2.3 THEN
	    //jeśli ustawiony bit startu z modbus i potwierdzone run napędu
	    %DB100.DBX33.1 := FALSE; // kasuj bit roskazu
	    ;
	  END_IF;
	  //Stop
	  //przekazanie bitu roskazu z bloku modbus rtu do bloku statusu napędu
	  IF %DB100.DBX33.5 THEN
	    %DB100.DBX2.4 := TRUE; //ustawienie bitu stop
	    ;
	  END_IF;
	  IF %DB100.DBX33.5 AND %DB100.DBX2.3 = FALSE THEN
	    //jeśli ustawiony bit stop z modbus i potwierdzone stop napędu
	    %DB100.DBX33.5 := FALSE; // kasuj bit roskazu
	    ;
	  END_IF;
	  
	END_REGION
	
	
	REGION //Drive Motor 3 ustaw na  Automat/Manual/Stop/Start
	  IF %DB100.DBX37.2 OR %DB100.DBX37.6 THEN
	    // przełączniki bistabilny każdy stan Hi powoduje zmianę przełącznika
	    #set_aut_man_M3 := TRUE; //ustawienie bitu start
	  ELSE
	    #set_aut_man_M3 := FALSE
	    ;
	  END_IF;
	  
	  IF %DB100.DBX4.0 = FALSE THEN
	    // przełącznik bistabilny
	    "R_TRIG_DB_AUT_M3"(CLK := #set_aut_man_M3,
	                       Q => #setTrig_M3);
	    ;
	  END_IF;
	  // przełącz na automat
	  IF #setTrig_M3 = TRUE AND %DB100.DBX37.2 = TRUE THEN
	    %DB100.DBX4.7 := TRUE;
	    ;
	  END_IF;
	  //przełącz na manual
	  IF #setTrig_M3 = TRUE AND %DB100.DBX37.6 = TRUE THEN
	    %DB100.DBX4.7 := FALSE;
	    ;
	  END_IF;
	  
	  IF (%DB100.DBX5.7 AND %DB100.DBX37.2) OR (%DB100.DBX5.7 = FALSE AND %DB100.DBX37.6) THEN
	    // Wyczyść całą zmienną
	    "dbHoldRegSlave_to_MT101".instConrol_ManAut_1 := 0;
	    // Kasowanie bitu 
	    %DB100.DBX37.2 := False;
	    %DB100.DBX37.6 := False;
	    ;
	  END_IF;
	  
	  // Start /
	  // przekazanie bitu roskazu z bloku modbus rtu do bloku statusu napędu
	  IF %DB100.DBX33.2 THEN
	    %DB100.DBX4.5 := TRUE; //ustawienie bitu start
	    ;
	  END_IF;
	  IF %DB100.DBX33.2 AND %DB100.DBX4.3 THEN
	    //jeśli ustawiony bit startu z modbus i potwierdzone run napędu
	    %DB100.DBX33.2 := FALSE; // kasuj bit roskazu
	    ;
	  END_IF;
	  //Stop
	  //przekazanie bitu roskazu z bloku modbus rtu do bloku statusu napędu
	  IF %DB100.DBX33.6 THEN
	    %DB100.DBX4.4 := TRUE; //ustawienie bitu stop
	    ;
	  END_IF;
	  IF %DB100.DBX33.6 AND %DB100.DBX4.3 = FALSE THEN
	    //jeśli ustawiony bit stop z modbus i potwierdzone stop napędu
	    %DB100.DBX33.6 := FALSE; // kasuj bit roskazu
	    ;
	  END_IF;
	  
	END_REGION
	
	
	REGION //Drive Motor 4 ustaw na  Automat/Manual/Stop/Start
	  IF %DB100.DBX37.3 OR %DB100.DBX37.7 THEN
	    // przełączniki bistabilny każdy stan Hi powoduje zmianę przełącznika
	    #set_aut_man_M4 := TRUE;
	  ELSE
	    #set_aut_man_M4 := FALSE
	    ;
	  END_IF;
	  
	  IF %DB100.DBX6.0 = FALSE THEN
	    // przełącznik bistabilny
	    "R_TRIG_DB_AUT_M4"(CLK := #set_aut_man_M4,
	                       Q => #setTrig_M4);
	    ;
	  END_IF;
	  
	  // przełącz na automat
	  IF #setTrig_M4 = TRUE AND %DB100.DBX37.3 = TRUE THEN
	    %DB100.DBX6.7 := TRUE;
	    ;
	  END_IF;
	  //przełącz na manual
	  IF #setTrig_M4 = TRUE AND %DB100.DBX37.7 = TRUE THEN
	    %DB100.DBX6.7 := FALSE;
	    ;
	  END_IF;
	  
	  IF (%DB100.DBX7.7 AND %DB100.DBX37.3) OR (%DB100.DBX7.7 = FALSE AND %DB100.DBX37.7) THEN
	    // Wyczyść całą zmienną
	    "dbHoldRegSlave_to_MT101".instConrol_ManAut_1 := 0;
	    // Kasowanie bitu 
	    %DB100.DBX37.3 := False;
	    %DB100.DBX37.7:= FALSE
	    ;
	  END_IF;
	  
	  // Start /
	  // przekazanie bitu roskazu z bloku modbus rtu do bloku statusu napędu
	  IF %DB100.DBX33.3 THEN
	    %DB100.DBX6.5 := TRUE; //ustawienie bitu start
	    ;
	  END_IF;
	  IF %DB100.DBX33.3 AND %DB100.DBX6.3 THEN
	    //jeśli ustawiony bit startu z modbus i potwierdzone run napędu
	    %DB100.DBX33.3 := FALSE; // kasuj bit roskazu
	    ;
	  END_IF;
	  //Stop
	  //przekazanie bitu roskazu z bloku modbus rtu do bloku statusu napędu
	  IF %DB100.DBX33.7 THEN
	    %DB100.DBX6.4 := TRUE; //ustawienie bitu stop
	    ;
	  END_IF;
	  IF %DB100.DBX33.7 AND %DB100.DBX6.3 = FALSE THEN
	    //jeśli ustawiony bit stop z modbus i potwierdzone stop napędu
	    %DB100.DBX33.7 := FALSE; // kasuj bit roskazu
	    ;
	  END_IF;
	  
	  
	END_REGION
	
	// Zasuwa Z1
	// 
	REGION //Drive Motor Z11 ustaw na  Automat/Manual/Otwieranie/Zamykanie
	  IF %DB100.DBX39.2 OR %DB100.DBX38.6 THEN
	    // przełączniki bistabilny każdy stan Hi powoduje zmianę przełącznika
	    #set_aut_man_Z11 := TRUE;
	  ELSE
	    #set_aut_man_Z11 := FALSE
	    ;
	  END_IF;
	  
	  IF %DB100.DBX28.0 = FALSE THEN
	    // przełącznik bistabilny
	    "R_TRIG_DB_AUT_Z11"(CLK := #set_aut_man_Z11,
	                        Q => #setTrig_Z11);
	    ;
	  END_IF;
	  //przełącz na automay
	  IF #setTrig_Z11 = TRUE AND %DB100.DBX39.2 = TRUE THEN
	    %DB100.DBX28.7 := TRUE;
	    ;
	  END_IF;
	  //przełącz na manual
	  IF #setTrig_Z11 = TRUE AND %DB100.DBX38.6 = TRUE THEN
	    %DB100.DBX28.7 := FALSE;
	    ;
	  END_IF;
	  
	  IF (%DB100.DBX29.7 AND %DB100.DBX39.2) OR (%DB100.DBX29.7 = FALSE AND %DB100.DBX38.6) THEN
	    // Wyczyść całą zmienną
	    "dbHoldRegSlave_to_MT101".instConrol_ManAut_2 := 0;
	    // Kasowanie bitu 
	    %DB100.DBX39.2 := False;
	    %DB100.DBX38.6 := FALSE
	    ;
	  END_IF;
	  
	  // Otwórz/
	  // przekazanie bitu roskazu z bloku modbus rtu do bloku statusu napędu
	  IF %DB100.DBX35.2 THEN
	    %DB100.DBX28.4 := %DB100.DBX35.2; //ustawienie bitu otwieranie
	    ;
	  END_IF;
	  IF %DB100.DBX35.2 AND %DB100.DBX29.1 THEN
	    //jeśli ustawiony bit otwierania z modbus i potwierdzone otwarcie 
	    %DB100.DBX35.2 := FALSE; // kasuj bit roskazu
	    ;
	  END_IF;
	  //Zamknij
	  //przekazanie bitu roskazu z bloku modbus rtu do bloku statusu napędu
	  IF %DB100.DBX34.6 THEN
	    %DB100.DBX28.5 := %DB100.DBX34.6; //ustawienie bitu zamykanie
	    ;
	  END_IF;
	  IF %DB100.DBX34.6 AND %DB100.DBX29.3 = FALSE THEN
	    //jeśli ustawiony bit zamykaniez modbus i potwierdzone zamknięcie 
	    %DB100.DBX34.6 := FALSE; // kasuj bit roskazu
	    ;
	  END_IF;
	  
	END_REGION
	
	
	
	
	
	(* 
	 ------------------------------------------------------------------------
	 
	Część obsługi PLC-2 obsługa czyszczenia zmiennych po odebraniu potwierdzeń  
	---------------------------------------------------------------------------
	*)
	
	
	
	
	
	
	
	
	
	
	
	
	
	
	
	
	
	
	
	
	
	
	
	  
	
	
	
	
END_FUNCTION_BLOCK

FUNCTION "08_C_ParsowanieDataTime_Zadanych_" : Void
TITLE = Persowanie danych data i time
{ S7_Optimized_Access := 'TRUE' }
AUTHOR : rtecmer
VERSION : 0.1
//Funkcja składa z wartości podanego czasu formie Real zmienne DTL przekazywane dale do układu sterowania zbiornikami i pompami

BEGIN
	(*
	//=============================================================================
	//(JZWiK S.A Radosław Tecmer)
	//(c)Copyright (2022) All Rights Reserved
	//-----------------------------------------------------------------------------
	//Testowane z:   (system docelowy z  FW 4.4)
	//Pakiet inżynierski:   TIA Portal (V16 Update 5)
	//Ograniczenia:  ( - )
	//Wymagania:  (minimalne S7-1200 CPU 1215C FW 4.2 .)
	//Funkcjonalnośc: (Persowanie danych wchodzących w formie Real do danych DTL
	                    Dane: czasy, sterowania zbiornikami i pracą pomp)
	//-----------------------------------------------------------------------------
	//Zmainy wprowadzone:
	//Wersja  Data       Osoba wprowadzająca zmiany - ekspert
	//01.00.00 09.03.2022 (Tecmer Radosław - twórca) Pieresza wersja 01.00.00
	//=============================================================================
	*)
	
	
	REGION start_napełnianie
	  // przekazanie z bloku SCADA do bloku danych programu PLC
	  "db10datablock".instHourStart_Filling.HOUR := INT_TO_USINT("dbHoldRegSlave_to_MT101".instHourStart_Filling);
	  "db10datablock".instHourStart_Filling.MINUTE := INT_TO_USINT("dbHoldRegSlave_to_MT101".instMinutStart_Filling);
	
	  
	END_REGION
	
	REGION Stop_napełnianie
	  // przekazanie z bloku SCADA do bloku danych programu PLC
	  "db10datablock".instHourStop_Filling.HOUR := INT_TO_USINT("dbHoldRegSlave_to_MT101".instHourStop_Filling);
	  "db10datablock".instHourStop_Filling.MINUTE := INT_TO_USINT("dbHoldRegSlave_to_MT101".instMinutStopt_Filling);
	  
	  
	END_REGION
	
	REGION Start_przetłaczanie_1
	  //
	  "db10datablock".instHourStart_City.HOUR := INT_TO_USINT("dbHoldRegSlave_to_MT101".instHourStart_City);
	  "db10datablock".instHourStart_City.MINUTE := INT_TO_USINT("dbHoldRegSlave_to_MT101".instMinutStart_City);
	 
	;
	  
	END_REGION
	
	REGION Stop_przetłaczanie_1
	  // przekazanie z bloku SCADA do bloku danych programu PLC
	  "db10datablock".instHourStop_City.HOUR := INT_TO_USINT("dbHoldRegSlave_to_MT101".instHourStop_City);
	  "db10datablock".instHourStop_City.MINUTE := INT_TO_USINT("dbHoldRegSlave_to_MT101".instMinutStopt_City);
	  
	
	  
	END_REGION
	
	REGION Start_dosilanie_1
	  // przekazanie z bloku SCADA do bloku danych programu PLC
	  "db10datablock".instHourStart_Replen.HOUR := INT_TO_USINT("dbHoldRegSlave_to_MT101".instHourStart_Replen);
	  "db10datablock".instHourStart_Replen.MINUTE := INT_TO_USINT("dbHoldRegSlave_to_MT101".instMinutStart_Replen);
	
	
	END_REGION
	
	REGION Stop_dosilanie_1
	  // przekazanie z bloku SCADA do bloku danych programu PLC
	  "db10datablock".instHourStop_Replen.HOUR := INT_TO_USINT("dbHoldRegSlave_to_MT101".instHourStop_Replen);
	  "db10datablock".instHourStop_Replen.MINUTE := INT_TO_USINT("dbHoldRegSlave_to_MT101".instMinutStopt_Replen);
	
	  // przekazanie do bloku danych wysyłanych 
	
	END_REGION
	
	
	
	
	
	
	
	
	
	
	
	
	
	
END_FUNCTION

FUNCTION "01_E_Clearing the given incorrect data" : Void
TITLE = Korekta błednego wpisu
{ S7_Optimized_Access := 'TRUE' }
AUTHOR : rtecmer
VERSION : 0.1
//Program kontroluje błedny wpis wartości poza granicą liczby określającej czas (godziny, minuty) W razie wpisania złej wartości wypełna komurkę zerami

BEGIN
	(*
	//=============================================================================
	//(JZWiK S.A Radosław Tecmer)
	//(c)Copyright (2022) All Rights Reserved
	//-----------------------------------------------------------------------------
	//Testowane z:   (system docelowy z  FW 4.4)
	//Pakiet inżynierski:   TIA Portal (V16 Update 5)
	//Ograniczenia:  ( - )
	//Wymagania:  (minimalne S7-1200 CPU 1215C FW 4.2 .)
	//Funkcjonalnośc: (Kontrola błednego wpisy wartości liczbowej czasu, wartości.
	                   Jeśli wartość poza zakresem wypełnieni komórki zerami)
	//-----------------------------------------------------------------------------
	//Zmainy wprowadzone:
	//Wersja  Data       Osoba wprowadzająca zmiany - ekspert
	//01.00.00 05.05.2022 (Tecmer Radosław - twórca) Pieresza wersja 01.00.00
	//=============================================================================
	*)
	
	
	
	
	
	//poziomy
	
	//napełnianie
	IF "dbHoldRegSlave_to_MT101".instLevelSetFilling < 0
	  OR "dbHoldRegSlave_to_MT101".instLevelSetFilling > 500
	  
	THEN
	  // ustaw
	  "dbHoldRegSlave_to_MT101".instLevelSetFilling := 300; 
	  
	  ;
	END_IF;
	
	//opróżnianie
	IF "dbHoldRegSlave_to_MT101".instLevelSetEmptying < 0
	  OR "dbHoldRegSlave_to_MT101".instLevelSetEmptying > 500
	  // porónaj jeśli wartość napełninia i opróżniania są takie same lub nie logiczne to ustaw domyślną
	  OR "dbHoldRegSlave_to_MT101".instLevelSetEmptying >= "dbHoldRegSlave_to_MT101".instLevelSetFilling
	 
	THEN
	  // ustaw
	  "dbHoldRegSlave_to_MT101".instLevelSetEmptying := 30;
	
	  ;
	END_IF;
	
	
	// czasy
	// 
	// napełnianie on
	IF "dbHoldRegSlave_to_MT101".instHourStart_Filling < 0
	  OR "dbHoldRegSlave_to_MT101".instHourStart_Filling > 23
	
	THEN
	  // ustaw
	  "dbHoldRegSlave_to_MT101".instHourStart_Filling := 0;
	
	  ;
	END_IF;
	
	IF "dbHoldRegSlave_to_MT101".instMinutStart_Filling < 0
	  OR "dbHoldRegSlave_to_MT101".instMinutStart_Filling > 60
	
	  THEN
	    // ustaw
	    "dbHoldRegSlave_to_MT101".instMinutStart_Filling := 0;
	
	
	    ;
	END_IF;
	
	// napełnianie off
	IF "dbHoldRegSlave_to_MT101".instHourStop_Filling < 0
	  OR "dbHoldRegSlave_to_MT101".instHourStop_Filling > 23
	
	THEN
	  // wypełnij zerami
	  "dbHoldRegSlave_to_MT101".instHourStop_Filling := 0;
	
	  ;
	END_IF;
	
	IF "dbHoldRegSlave_to_MT101".instMinutStopt_Filling < 0
	  OR "dbHoldRegSlave_to_MT101".instMinutStopt_Filling > 60
	
	THEN
	  // wypełnij zerami
	  "dbHoldRegSlave_to_MT101".instMinutStopt_Filling := 0;
	
	  ;
	END_IF;
	
	
	
	
	
END_FUNCTION

FUNCTION "04_A_IN" : Void
TITLE = Mapping control room inputs
{ S7_Optimized_Access := 'TRUE' }
AUTHOR : rtecmer
VERSION : 0.1
//Sprawdzanie wejść sterowniak i przekazanie sygnałów 
   VAR_TEMP 
      ruchZ11 : Bool;   // ruch zasuwy
   END_VAR


BEGIN
	
	(*
	//=============================================================================
	//(JZWiK S.A Radosław Tecmer)
	//(c)Copyright (2021) All Rights Reserved
	//-----------------------------------------------------------------------------
	//Testowane z:   (system docelowy z  FW 4.4)
	//Pakiet inżynierski:   TIA Portal (V14 Sp1 Update 9)
	//Ograniczenia:  ( - )
	//Wymagania:  (minimalne S7-1200 CPU 1215C FW 4.2 .)
	//Funkcjonalnośc: (Mapowanie wejść sterownika
	//                 Sprawdzanie wejść sterowniak i przekazanie sygnałów )
	//-----------------------------------------------------------------------------
	//Zmainy wprowadzone:
	//Wersja  Data       Osoba wprowadzająca zmiany - ekspert
	//01.00.00 19.01.2022 (Tecmer Radosław - twórca) Pieresza wersja 01.00.00
	//=============================================================================
	*)
	
	// Pompy
	REGION Tryb sterowania Pompami
	  // ustawienie znacznika tryb pracy z systemu 1= Aut 0=REM
	  "inputRem_P1-P4" := "I0.4":P;
	  "IsRem" := "inputRem_P1-P4";
	  
	END_REGION
	
	
	
	// POMPA P1
	"IEC_Timer_P1_ready_DB".TOF(IN := "I0.0":P , // histereza na awarię
	                            PT := T#12S,
	                            Q => "inputReadyP1");
	                            
	
	
	"inputRunF_P1" := "I0.5":P;
	"inputRunS_P1" := "I0.6":P;
	
	// POMPA P2
	"IEC_Timer_P2_ready_DB".TOF(IN:="I0.1":P, // histereza na awarię
	                            PT:=T#10S,
	                            Q => "inputReadyP2" );
	
	
	"inputRunF_P2" := "I0.7":P;
	"inputRunS_P2" := "I1.0":P;
	
	// POMPA P3
	"IEC_Timer_P3_ready_DB".TOF(IN:="I0.2":P, // histereza na awarię
	                            PT:=T#10S,
	                            Q=>"inputReadyP3");
	
	
	"inputRunF_P3" := "I1.1":P;
	"inputRunS_P3" := "I1.2":P;
	
	//---------------
	
	
	// STOP AWARIA PRZYCISK
	"INPUTstopAccident_Pompy" := "I1.4":P;
	
	
	//Zasuwa Z1
	REGION Z11
	  IF "inputOtwartaZ11" = FALSE AND "inputOtwartaZ11" = FALSE THEN
	    // ustaw flagę ruch
	    #ruchZ11 := TRUE;
	  ELSE
	  #ruchZ11 := FALSE;
	    ;
	  END_IF;
	  
	  // ZASUWY Z1
	  "inputREM_ZASUWY" := "I2.1":P;
	  
	  "inputRuchZ11" := #ruchZ11;
	  "inputAwariaMomentZ11" := "I2.0":P; // gotowość
	  "inputOtwartaZ11" := "I2.2":P;
	  "inputZamkniętaZ11" := "I2.3":P;
	
	  
	END_REGION
	
	
	
	// ######################
	// Szafa RS Zasilanie OK
	"inputpowerOK_RS" := "I0.3":P;
	"Is_PowerRS5_OK" := "inputpowerOK_RS";
	// #########################
	
	// Gotowość P1
	REGION Gotowość P1
	  // Gdy brak sygnału na wejściu GOTO lub w statusie ustawiony bit awarii
	  // to brak gotowości
	  IF "inputReadyP1" = FALSE OR "bitH_Alarm_P1"= TRUE THEN
	    "IsReady_P1" := FALSE;
	  ELSE
	    "IsReady_P1" := TRUE;
	  END_IF;
	  
	END_REGION
	
	// Gotowość P2
	REGION Gotowość P2
	  // Gdy brak sygnału na wejściu GOTO lub w statusie ustawiony bit awarii
	  // to brak gotowości
	  IF "inputReadyP2" = FALSE OR "bitH_Alarm_P2" = TRUE THEN
	    "IsReady_P2" := FALSE;
	  ELSE
	    "IsReady_P2" := TRUE;
	  END_IF;
	  
	END_REGION
	
	// Gotowość P3
	REGION Gotowość P3
	  // Gdy brak sygnału na wejściu GOTO lub w statusie ustawiony bit awarii
	  // to brak gotowości
	  IF "inputReadyP3" = FALSE OR "bitH_Alarm_P3" = TRUE  THEN
	    "IsReady_P3" := FALSE;
	  ELSE
	    "IsReady_P3" := TRUE;
	  END_IF;
	  
	END_REGION
	
	
	// Gotowość P4  - pompy brak, zestaw 3 pomp
	"IsReady_P4" := FALSE;
	
	
	// Gotowość falownika
	"inputready_Inverter_P1-P4" := "I1.5":P;
	
	IF "inputready_Inverter_P1-P4"  THEN
	  // Ustaw gotowość
	  "IsReady_Inverter" :=TRUE;
	ELSE
	  "IsReady_Inverter" := FALSE;
	  ;
	END_IF;
	
	REGION Praca falownika
	  "inputrunInverter_" := "I1.3":P;
	  "IsRunInverter1" := "inputrunInverter_";
	  
	END_REGION
	
	REGION Potwierdzenia pracy falownik, sieć
	  "IsRunInverter_P1" := "inputRunF_P1";
	  "IsRunNetwork_P1" := "inputRunS_P1";
	  "IsRunInverter_P2" := "inputRunF_P2";
	  "IsRunNetwork_P2" := "inputRunS_P2";
	  "IsRunInverter_P3" := "inputRunF_P3";
	  "IsRunNetwork_P3" := "inputRunS_P3";
	
	  
	END_REGION
	
	
	
	REGION Pompa P1
	  // Sygnał Run P1
	  IF "IsRunInverter_P1" OR "IsRunNetwork_P1" THEN
	    "IsRun_P1" := TRUE;
	  ELSE
	    "IsRun_P1" := FALSE;
	  END_IF;
	  
	END_REGION
	
	REGION Pompa P2
	  // Sygnał Run P2
	  IF "IsRunInverter_P2" OR "IsRunNetwork_P2" THEN
	    "IsRun_P2" := TRUE;
	  ELSE
	    "IsRun_P2" := FALSE;
	  END_IF;
	  
	END_REGION
	
	
	REGION Pompa P3
	  // Sygnał Run P3
	  IF "IsRunInverter_P3" OR "IsRunNetwork_P3" THEN
	    "IsRun_P3" := TRUE;
	  ELSE
	    "IsRun_P3" := FALSE;
	  END_IF;
	  
	END_REGION
	
	
	
	
	
	
	
	
	
	
END_FUNCTION

FUNCTION_BLOCK "06_M_Byte status Z11 Z12"
TITLE = Calculation Byte Status M1-M4
{ S7_Optimized_Access := 'TRUE' }
AUTHOR : rtecmer
VERSION : 0.1
//Byte określający ile napędów dostępnych. Wykorzystywany do blokowania przełączenia na sieć ostatniej dostępnej pompy.

BEGIN
	(*
	//=============================================================================
	//(JZWiK S.A Radosław Tecmer)
	//(c)Copyright (2021) All Rights Reserved
	//-----------------------------------------------------------------------------
	//Testowane z:   (system docelowy z  FW 4.4)
	//Pakiet inżynierski:   TIA Portal (V14 Sp1 Update 9)
	//Ograniczenia:  ( - )
	//Wymagania:  (minimalne S7-1200 CPU 1215C FW 4.2 .)
	//Funkcjonalnośc: (Byte statusu napędów Z11 Z12 Zasuwy )
	//-----------------------------------------------------------------------------
	//Zmainy wprowadzone:
	//Wersja  Data       Osoba wprowadzająca zmiany - ekspert
	//01.00.00 17.11.2021 (Tecmer Radosław - twórca) Pieresza wersja 01.00.00
	//=============================================================================
	*)
	
	
	
	
	
	REGION przekazanie satusu Z11 Z12  do znacznika
	  //przekazanie
	  // Z11 Przekazanie Byte H ststusu do Byte znacznika 
	  "Byte_Status_Z11" := %DB100.DBB29;
	
	
	  
	  
	END_REGION
	
END_FUNCTION_BLOCK

FUNCTION_BLOCK "02_R_TimeSyn_PLC_To_HMI"
{ S7_Optimized_Access := 'FALSE' }
VERSION : 0.1
   VAR_OUTPUT 
      PLC_RD_LOC_T {InstructionName := 'DTL'; LibVersion := '1.0'} : DTL;
      PLC_RD_SYS_T {InstructionName := 'DTL'; LibVersion := '1.0'} : DTL;
   END_VAR

   VAR_IN_OUT 
      AreaPointer_JobMailbox : Array[0..3] of Word;
      SetTime : Bool;
      SetDate : Bool;
   END_VAR

   VAR 
      Func_RD_LOC_T {InstructionName := 'DTL'; LibVersion := '1.0'} : DTL;
      Ret_Val_RD_LOC_T : Int;
      BCD_Hour : Word;
      BCD_Minute : Word;
      BCD_Second : Word;
      BCD_Weekdday : Word;
      BCD_Day : Word;
      BCD_Month : Word;
      BCD32_Year : DWord;
      BCD16_Year : Word;
      STEP1 : Bool;
      STEP2 : Bool;
      STEP3 : Bool;
      STEP10 : Bool;
      STEP11 : Bool;
      STEP12 : Bool;
      Func_RD_SYS_T {InstructionName := 'DTL'; LibVersion := '1.0'} : DTL;
      Ret_Val_RD_SYS_T : Int;
   END_VAR


BEGIN
	//SIMATIC S7-1200 / 1500
	//
	
	//Odczyt aktualnego czasu PLC // Odczyt aktualnego czasu PLC
	#Ret_Val_RD_LOC_T := RD_LOC_T(#Func_RD_LOC_T);
	#PLC_RD_LOC_T := (#Func_RD_LOC_T);
	#Ret_Val_RD_SYS_T := RD_SYS_T(#Func_RD_SYS_T);
	#PLC_RD_SYS_T := (#Func_RD_SYS_T);
	
	
	//***Czas transmisja
	//Step 1
	//Zacznij, jeśli job mailmox  ma wartość zero.    
	IF #SetTime AND (#AreaPointer_JobMailbox[0] = 0) THEN
	    
	    //Parameter 1-3: Mit Null "0" vorbelegen //Parameters 1-3: Preassign with zero "0"
	    #AreaPointer_JobMailbox[1] := 0;
	    #AreaPointer_JobMailbox[2] := 0;
	    #AreaPointer_JobMailbox[3] := 0;
	    
	    #SetTime := false;
	    #STEP2 := true;
	    
	END_IF;
	
	//Step 2
	//plc job 14 - assign parameter
	IF #STEP2 THEN
	    
	    //Convert USInt to BCD format (plc job 14 need bcd format)
	    #BCD_Hour := INT_TO_BCD16(#Func_RD_LOC_T.HOUR);
	    #BCD_Minute := INT_TO_BCD16(#Func_RD_LOC_T.MINUTE);
	    #BCD_Second := INT_TO_BCD16(#Func_RD_LOC_T.SECOND);
	    
	    //Parameter
	    #AreaPointer_JobMailbox[1].%B0 := #BCD_Hour.%B0;
	    #AreaPointer_JobMailbox[2].%B1 := #BCD_Minute.%B0;
	    #AreaPointer_JobMailbox[2].%B0 := #BCD_Second.%B0;
	    
	    //plc job 14
	    #AreaPointer_JobMailbox[0] := 14;
	    
	    #STEP2 := FALSE;
	    
	END_IF;
	
	
	//****Data przesłania
	//Step 10
	//Start, if job mailbox are zero.    
	IF #SetDate AND (#AreaPointer_JobMailbox[0] = 0) THEN
	    
	    //Parameters 1-3: Preassign with zero "0"
	    #AreaPointer_JobMailbox[1] := 0;
	    #AreaPointer_JobMailbox[2] := 0;
	    #AreaPointer_JobMailbox[3] := 0;
	    
	    #SetDate := false;
	    #STEP11 := true;
	    
	END_IF;
	
	//Step 11
	//plc job 15 - assign parameter
	IF #STEP11 THEN
	    
	    //Convert USInt to BCD  (plc job 15 need bcd format)
	    #BCD_Weekdday := INT_TO_BCD16(#Func_RD_LOC_T.WEEKDAY);
	    #BCD_Day := INT_TO_BCD16(#Func_RD_LOC_T.DAY);
	    #BCD_Month := INT_TO_BCD16(#Func_RD_LOC_T.MONTH);
	    #BCD32_Year := DINT_TO_BCD32(#Func_RD_LOC_T.YEAR);
	    // convert BCD32 to BCD16
	    #BCD16_Year := DWORD_TO_WORD(#BCD32_Year);
	    
	    //Parameter
	    #AreaPointer_JobMailbox[1].%B0 := #BCD_Weekdday.%B0;
	    #AreaPointer_JobMailbox[2].%B1 := #BCD_Day.%B0;
	    #AreaPointer_JobMailbox[2].%B0 := #BCD_Month.%B0;
	    #AreaPointer_JobMailbox[3].%B1 := #BCD16_Year.%B0;
	    
	    //plc job 15
	    #AreaPointer_JobMailbox[0] := 15;
	    
	    #STEP11 := FALSE;
	    
	END_IF;
	
	
END_FUNCTION_BLOCK

FUNCTION "06_M_Switch of signal source of pressure" : Void   // FC5, LAD
{ S7_Optimized_Access := 'TRUE' }
AUTHOR : rtecmer
VERSION : 0.1
// Przęłączanie sygnału źródła ciśnienia zależnie od wybranej strategi: 
// 0- wyłączone, 1- Dosilanie, 2- Przetłączanie, 3- Automat, 4- Ręczne
// stored: AutoNumber true, IsIECCheckEnabled false, SetENOAutomatically false, UDAEnableTagReadback false
   VAR_TEMP   // added for the SCL form of the ladder/FBD networks
      _w1 : Bool;
   END_VAR
BEGIN

REGION Network 1: Filtr Kolmana
   // "switch_kolman" - jeśli 1 to wyłączony jeśli 0 - załączony
END_REGION

REGION Network 2: PV do regulatora PI
   // Podajemy sygnał do PI PV
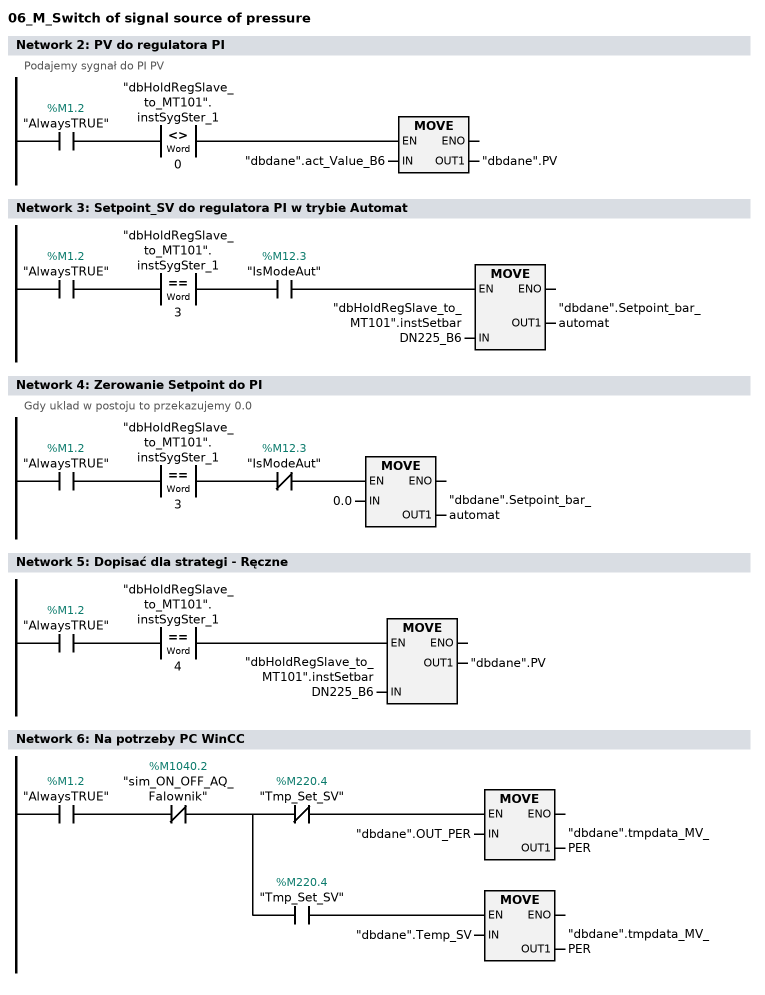
   RUNG wire#powerrail
      Contact( "AlwaysTRUE" )
      { S7_Templates := "SrcType := Word" } NE_Contact(in1 := "dbHoldRegSlave_to_MT101".instSygSter_1, in2 := 0)
      Move(in := "dbdane".act_Value_B6, out1 => "dbdane".PV)
   END_RUNG
   // the same network as SCL:
   IF "AlwaysTRUE" AND ("dbHoldRegSlave_to_MT101".instSygSter_1 <> 0) THEN
       "dbdane".PV := "dbdane".act_Value_B6;
   END_IF;
END_REGION

REGION Network 3: Setpoint_SV do regulatora PI w trybie Automat
   RUNG wire#powerrail
      Contact( "AlwaysTRUE" )
      { S7_Templates := "SrcType := Word" } EQ_Contact(in1 := "dbHoldRegSlave_to_MT101".instSygSter_1, in2 := 3)
      Contact( "IsModeAut" )
      Move(in := "dbHoldRegSlave_to_MT101".instSetbarDN225_B6, out1 => "dbdane".Setpoint_bar_automat)
   END_RUNG
   // the same network as SCL:
   IF "AlwaysTRUE" AND ("dbHoldRegSlave_to_MT101".instSygSter_1 = 3) AND "IsModeAut" THEN
       "dbdane".Setpoint_bar_automat := "dbHoldRegSlave_to_MT101".instSetbarDN225_B6;
   END_IF;
END_REGION

REGION Network 4: Zerowanie Setpoint do PI
   // Gdy uklad w postoju to przekazujemy 0.0
   RUNG wire#powerrail
      Contact( "AlwaysTRUE" )
      { S7_Templates := "SrcType := Word" } EQ_Contact(in1 := "dbHoldRegSlave_to_MT101".instSygSter_1, in2 := 3)
      I_Contact( "IsModeAut" )
      Move(in := 0.0, out1 => "dbdane".Setpoint_bar_automat)
   END_RUNG
   // the same network as SCL:
   IF "AlwaysTRUE" AND ("dbHoldRegSlave_to_MT101".instSygSter_1 = 3) AND NOT "IsModeAut" THEN
       "dbdane".Setpoint_bar_automat := 0.0;
   END_IF;
END_REGION

REGION Network 5: Dopisać dla strategi - Ręczne
   RUNG wire#powerrail
      Contact( "AlwaysTRUE" )
      { S7_Templates := "SrcType := Word" } EQ_Contact(in1 := "dbHoldRegSlave_to_MT101".instSygSter_1, in2 := 4)
      Move(in := "dbHoldRegSlave_to_MT101".instSetbarDN225_B6, out1 => "dbdane".PV)
   END_RUNG
   // the same network as SCL:
   IF "AlwaysTRUE" AND ("dbHoldRegSlave_to_MT101".instSygSter_1 = 4) THEN
       "dbdane".PV := "dbHoldRegSlave_to_MT101".instSetbarDN225_B6;
   END_IF;
END_REGION

REGION Network 6: Na potrzeby PC WinCC
   RUNG wire#powerrail
      Contact( "AlwaysTRUE" )
      I_Contact( "sim_ON_OFF_AQ_Falownik" )
      wire#w1
      I_Contact( "Tmp_Set_SV" )
      { S7_GenerateENO := "TRUE" } Move(in := "dbdane".OUT_PER, out1 => "dbdane".tmpdata_MV_PER)
   END_RUNG
   RUNG wire#w1
      Contact( "Tmp_Set_SV" )
      { S7_GenerateENO := "TRUE" } Move(in := "dbdane".Temp_SV, out1 => "dbdane".tmpdata_MV_PER)
   END_RUNG
   // the same network as SCL:
   #_w1 := "AlwaysTRUE" AND NOT "sim_ON_OFF_AQ_Falownik";
   IF #_w1 AND NOT "Tmp_Set_SV" THEN "dbdane".tmpdata_MV_PER := "dbdane".OUT_PER; END_IF;
   IF #_w1 AND "Tmp_Set_SV" THEN "dbdane".tmpdata_MV_PER := "dbdane".Temp_SV; END_IF;
END_REGION
END_FUNCTION

FUNCTION "08_M_Read_Inverter ModbusRTU" : Void   // FC22, LAD
TITLE = Modbus RTU Inverter
{ S7_Optimized_Access := 'TRUE' }
VERSION : 0.1
// Cykliczna komunikacja Modbus RTU Falownik
// stored: AutoNumber true, IsIECCheckEnabled false, SetENOAutomatically false, UDAEnableTagReadback false
   VAR_TEMP   // added for the SCL form of the ladder/FBD networks
      _w1 : Bool;
      _w2 : Bool;
   END_VAR
BEGIN

REGION Network 2: ARESS 26-----------------------------------------------------
END_REGION

REGION Network 3: MODBUS RTU adress 26*****step 1: read from inverter control words
   // Pobieranie słowa controlnego
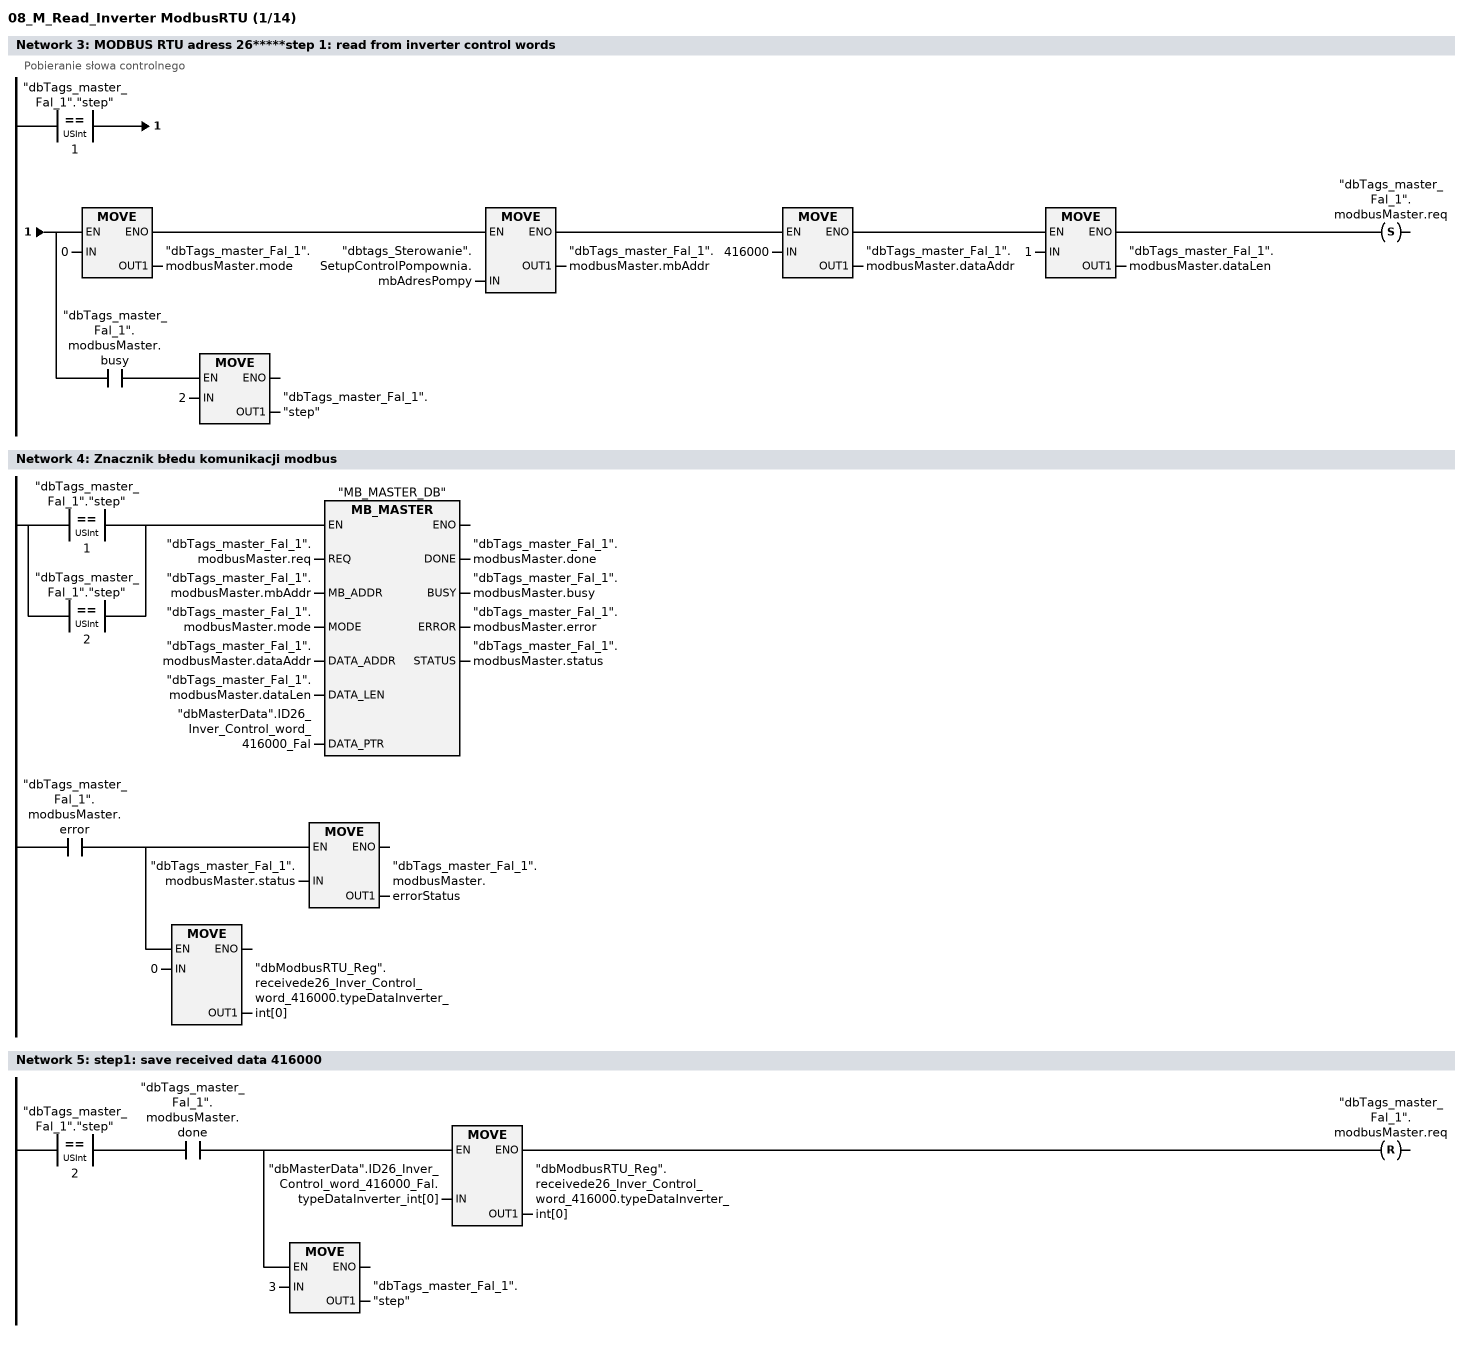
   RUNG wire#powerrail
      { S7_Templates := "SrcType := USInt" } EQ_Contact(in1 := "dbTags_master_Fal_1"."step", in2 := 1)
      wire#w1
      { S7_GenerateENO := "TRUE" } Move(in := 0, out1 => "dbTags_master_Fal_1".modbusMaster.mode)
      Move(in := "dbtags_Sterowanie".SetupControlPompownia.mbAdresPompy, out1 => "dbTags_master_Fal_1".modbusMaster.mbAddr)
      { S7_GenerateENO := "TRUE" } Move(in := 416000, out1 => "dbTags_master_Fal_1".modbusMaster.dataAddr)
      Move(in := 1, out1 => "dbTags_master_Fal_1".modbusMaster.dataLen)
      S_Coil( "dbTags_master_Fal_1".modbusMaster.req )
   END_RUNG
   RUNG wire#w1
      Contact( "dbTags_master_Fal_1".modbusMaster.busy )
      { S7_GenerateENO := "TRUE" } Move(in := 2, out1 => "dbTags_master_Fal_1"."step")
   END_RUNG
   // the same network as SCL:
   // ENO of a box is taken as its EN; it also drops when the box reports an error
   #_w1 := "dbTags_master_Fal_1"."step" = 1;
   IF #_w1 THEN
       "dbTags_master_Fal_1".modbusMaster.mode := 0;
       "dbTags_master_Fal_1".modbusMaster.mbAddr := "dbtags_Sterowanie".SetupControlPompownia.mbAdresPompy;
       "dbTags_master_Fal_1".modbusMaster.dataAddr := 416000;
       "dbTags_master_Fal_1".modbusMaster.dataLen := 1;
       "dbTags_master_Fal_1".modbusMaster.req := TRUE;
   END_IF;
   IF #_w1 AND "dbTags_master_Fal_1".modbusMaster.busy THEN "dbTags_master_Fal_1"."step" := 2; END_IF;
END_REGION

